   (*=================================================================================*)
   (* AM03_2   ---   Read Status + Send Control / Read Voltage + Current *)
   (*=================================================================================*)
   IF #Block2Size > 0 THEN
       // Read Total current and calculate it
       IF #C_Block2_TotalCurrent > 0 THEN
           (*Read Data*)
           #iError := DPRD_DAT(LADDR := #C_Block2_TotalCurrent, RECORD => #Current);
           (*Calculate Value*)
           #CalcValue := #Current[1];
           #CalcValue := SHL(IN := #CalcValue, N := 8);
           #O_Block2TotalCurrent := (#CalcValue + #Current[0]) / 100;
       END_IF;
       (*Status And Control*)
       IF #C_Block2_StatusControl > 0 THEN
           (*Read Inputs*)
           #iError := DPRD_DAT(LADDR := #C_Block2_StatusControl, RECORD => #Status);
           (*Take it over to the Datastructure*)
           FOR #iCount := 1 TO 32 DO
               IF #iCount <= #Block2Size * 2 THEN //WDL changed C_Block1Size by C_Block2Size
                   IF "SimulationActive" THEN
                       "NotUsedBool" := False;
                     ELSE
                       #IO_ETAFuseData.DataCPC20.Fuse[#iCount + 32].Status := #Status[#iCount]; (*Read Status*)
                   END_IF;
                   #Control[#iCount] := #IO_ETAFuseData.DataCPC20.Fuse[#iCount + 32].Control; (*Write control to the buffer*)
               ELSE
                   #IO_ETAFuseData.DataCPC20.Fuse[#iCount + 32].Status := 255; (*Read Status*)
                   #Control[#iCount] := 0; (*Write control to the buffer*)
               END_IF;
           END_FOR;
           (*Write outputs to the CPC*)
           #iError := DPWR_DAT(LADDR := #C_Block2_StatusControl, RECORD := #Control);
       END_IF;
       (*Measurement preperation*)
       IF #"C_Block2_MeasurementU/I" > 0 THEN
           (*Read measurenets values*)
           #iError := DPRD_DAT(LADDR := #"C_Block2_MeasurementU/I", RECORD => #UI);
           (*Create Measurements*)
           FOR #iCount := 1 TO 32 DO
               (*Calculate new Adress*)
               #iCalcAddress := ((#iCount - 1) * 4);
               IF #iCount <= #Block2Size * 2 THEN
                   (*Calculate current and take it over to the Datastructure*)
                   #CalcValue := #UI[#iCalcAddress + 1]; (*-2*)
                   #CalcValue := SHL(IN := #CalcValue, N := 8);
                   #IO_ETAFuseData.DataCPC20.Fuse[#iCount + 32].Current := INT_TO_REAL(#CalcValue + #UI[#iCalcAddress]) / 100; (*-3*)
                   (*Calculate voltage and take it over to the Datastructure*)
                   #CalcValue := #UI[#iCalcAddress + 3];
                   #CalcValue := SHL(IN := #CalcValue, N := 8); (*-0*)
                   #IO_ETAFuseData.DataCPC20.Fuse[#iCount + 32].Voltage := INT_TO_REAL(#CalcValue + #UI[#iCalcAddress + 2]) / 100; (*-1*)
               ELSE
                   #IO_ETAFuseData.DataCPC20.Fuse[#iCount + 32].Current := 0; (*-3*)
                   #IO_ETAFuseData.DataCPC20.Fuse[#iCount + 32].Voltage := 0; (*-1*)
               END_IF;
           END_FOR;
       END_IF;
   END_IF;

   (*=================================================================================*)
   (*AM03_1 & AM03_2   ---   Read Nominal Current *)    
   (*=================================================================================*)
   //HMI Command - Cancel Read nominal current
   IF #I_CancelReadNomCurr OR "SimulationActive" THEN
       #iCountGet := 1000;
   END_IF;

   CASE #iCountGet OF
       0: IF (#InitNominalCurrent OR #I_ReadNomCurr OR #I_NewShift) AND NOT #NonCyclicCommunication.ReadNomCurrActive AND NOT "SimulationActive" THEN
               IF (#C_Block1_TotalCurrent > 0) THEN
                   #iCountNominalCurrent := 1; // Init Value
                   #ChannelNumber := 1; // Init Value
                   #HardwareID := #C_Block1_TotalCurrent; // Init Value
                   #NonCyclicCommunication.ReadNomCurrActive := True;
                   #iCountGet := 10;
               END_IF;

               IF (#C_Block1_TotalCurrent = 0) AND (#C_Block2_TotalCurrent > 0) THEN
                   #iCountNominalCurrent := 33; // Init Value
                   #ChannelNumber := 1; // Init Value
                   #HardwareID := #C_Block2_TotalCurrent; // Init Value
                   #NonCyclicCommunication.ReadNomCurrActive := True;
                   #iCountGet := 10;
               END_IF;

               IF (#C_Block1_TotalCurrent = 0) AND (#C_Block2_TotalCurrent = 0) THEN
                   #Get.bGetData := False;
                   #iCountGet := 1000;
               END_IF;
           END_IF;
       10: // Set Parameter to read a channel and start it
           IF NOT #C_Config.Fuse[#iCountNominalCurrent].Used THEN
               #iCountNominalCurrent := #iCountNominalCurrent + 1;
               #ChannelNumber := #ChannelNumber + 1;
               #IO_ETAFuseData.DataCPC20.Fuse[#iCountNominalCurrent].NominalCurrent := 0;
               #iCountGet := 100;
           ELSE
               #Get.diIndex := (#ChannelNumber * 100) + 1; // Channel Number * Factor for Parameter + Index
               #Get.uiMlen := 8;
               #Get.bGetData := True; (*Read Data*)
               #iCountGet := 20;
           END_IF;

           IF (#iCountNominalCurrent >= 64) THEN
               #iCountGet := 1000;
           END_IF;
       20: (*reading is active*)
           IF #Get.bBusy OR #Get.bError THEN
               #Get.bGetData := false; (*Edge to read is enough*)
               #iCountGet := 30;
           END_IF;
       30: (*Evaluate data, stop reading, set message in case of error*)
           IF NOT #Get.bBusy THEN
               IF #Get.bValid THEN
                   #IO_ETAFuseData.DataCPC20.Fuse[#iCountNominalCurrent].NominalCurrent := #Get.DataByte[1] - 16#A0;
                   #iCountGet := 100;
               ELSE
                   #iCountGet := 10;
               END_IF;
           END_IF;
       100: // check for next channel
           IF (#iCountNominalCurrent >= 32) AND (#iCountNominalCurrent < 64) THEN
               #HardwareID := #C_Block2_TotalCurrent;
               #iCountNominalCurrent := #iCountNominalCurrent + 1;
               #ChannelNumber := #ChannelNumber + 1;
               #iCountGet := 10;
           END_IF;

           IF #iCountNominalCurrent < 32 THEN
               #HardwareID := #C_Block1_TotalCurrent;
               #iCountNominalCurrent := #iCountNominalCurrent + 1;
               #ChannelNumber := #ChannelNumber + 1;
               #iCountGet := 10;
           END_IF;

           IF (#iCountNominalCurrent = 33) THEN
               #ChannelNumber := 1;
           END_IF;

           IF (#iCountNominalCurrent >= 64) THEN
               #iCountGet := 1000;
           END_IF;
       1000: // End
           #InitNominalCurrent := False;
           #NonCyclicCommunication.ReadNomCurrActive := False;
           #iCountGet := 0;
   END_CASE;

   // Reading of nominal current is active
   #O_ReadNomCurrActive := #NonCyclicCommunication.ReadNomCurrActive;
   #O_ReadNomCurrFuseNr := #iCountNominalCurrent;

   // Overtime Reading of nominal current
   #T_ReadNomCurr(IN:= #O_ReadNomCurrActive,
                  PT:= T#60s);

   #O_AlarmReadNomCurr := #T_ReadNomCurr.Q;

   // Call noncyclic communication
   #RDREC_FB(REQ := #Get.bGetData,
             ID := #HardwareID,
             INDEX := #Get.diIndex,
             MLEN := #Get.uiMlen,
             VALID => #Get.bValid,
             BUSY => #Get.bBusy,
             ERROR => #Get.bError,
             STATUS => #Get.dwState,
             LEN => #Get.uilen,
             RECORD := #Get.DataByte);

   (*=================================================================================*)
   (* Fill-in/Clear Information *)    
   (*=================================================================================*)
   FOR #iCount := 1 TO 64 DO
       IF #C_Config.Fuse[#iCount].Used THEN
           #IO_ETAFuseData.ForHMICPC20.Fuse[#iCount].Used := True;
           #H_ETAFuseCPC20PN.H_ForHMI.ChannelInfo[#iCount].Name := #C_Config.Fuse[#iCount].Name;
           #H_ETAFuseCPC20PN.H_ForHMI.ChannelInfo[#iCount].Description := #C_Config.Fuse[#iCount].Description;
           #H_ETAFuseCPC20PN.H_ForHMI.ChannelInfo[#iCount].Current := #IO_ETAFuseData.DataCPC20.Fuse[#iCount].Current;
           #H_ETAFuseCPC20PN.H_ForHMI.ChannelInfo[#iCount].NominalCurrent := #IO_ETAFuseData.DataCPC20.Fuse[#iCount].NominalCurrent;
       ELSE
           #IO_ETAFuseData.DataCPC20.Fuse[#iCount] := #EmptyDataCPC20;
           #IO_ETAFuseData.DataCPC20.Fuse[#iCount].Status := 255;

           #IO_ETAFuseData.ForHMICPC20.Fuse[#iCount] := #EmptyForHMIFuse;

           #H_ETAFuseCPC20PN.H_ForHMI.Fuse[#iCount] := #EmptyForHMIFuse;
           #H_ETAFuseCPC20PN.H_ForHMI.ChannelInfo[#iCount] := #EmptyForHMIChannelInfo;
           #H_ETAFuseCPC20PN.H_ForHMI.ChannelInfo[#iCount].Name := 'Not exist';
       END_IF;
   END_FOR;

   #H_ETAFuseCPC20PN.H_ForHMI.Fuse := #IO_ETAFuseData.ForHMICPC20.Fuse;
END_FUNCTION_BLOCK

FUNCTION_BLOCK "L10Alarm"   // FB1410, FBD
TITLE = L10Alarm
{ S7_Optimized_Access := 'FALSE' }
AUTHOR : VCC
FAMILY : AlarmHnd
NAME : 10Alarm
VERSION : 1.0
// ================================================================================
// This module is used everywhere 10 alarms has to be generated when one 
// (security) corresponding input becomes True.
// All alarms can be True only when the corresponding input Enable Alarm is also 
// True.
// When the conditions to generate the alarm is disappear, a boolean (one per 
// alarm) available to inform the upper level that the corresponding alarm can be 
// reset. All alarms are reset by means of the AlarmResetPB signal.
// ================================================================================
// stored: AutoNumber false, IsIECCheckEnabled false, SetENOAutomatically False, UDAEnableTagReadback false
   VAR_INPUT
      I_Input1 { ExternalAccessible := 'False'; ExternalVisible := 'False'; ExternalWritable := 'False'} : Bool;   // Input alarm 1
      I_AlarmClass1 { ExternalAccessible := 'False'; ExternalVisible := 'False'; ExternalWritable := 'False'} : Char;   // Alarm class -> A - B - C - D or E
      I_EnableAlarm1 { ExternalAccessible := 'False'; ExternalVisible := 'False'; ExternalWritable := 'False'} : Bool := TRUE;   // Enable alarm 1 from upper level
      I_Invisible1 { ExternalAccessible := 'False'; ExternalVisible := 'False'; ExternalWritable := 'False'} : Bool;   // Invisible 1
      I_Input2 { ExternalAccessible := 'False'; ExternalVisible := 'False'; ExternalWritable := 'False'} : Bool;   // Input alarm 2
      I_AlarmClass2 { ExternalAccessible := 'False'; ExternalVisible := 'False'; ExternalWritable := 'False'} : Char;   // Alarm class -> A - B - C - D or E
      I_EnableAlarm2 { ExternalAccessible := 'False'; ExternalVisible := 'False'; ExternalWritable := 'False'} : Bool := TRUE;   // Enable alarm 2 from upper level
      I_Invisible2 { ExternalAccessible := 'False'; ExternalVisible := 'False'; ExternalWritable := 'False'} : Bool;   // Invisible 2
      I_Input3 { ExternalAccessible := 'False'; ExternalVisible := 'False'; ExternalWritable := 'False'} : Bool;   // Input alarm 3
      I_AlarmClass3 { ExternalAccessible := 'False'; ExternalVisible := 'False'; ExternalWritable := 'False'} : Char;   // Alarm class -> A - B - C - D or E
      I_EnableAlarm3 { ExternalAccessible := 'False'; ExternalVisible := 'False'; ExternalWritable := 'False'} : Bool := TRUE;   // Enable alarm 3 from upper level
      I_Invisible3 { ExternalAccessible := 'False'; ExternalVisible := 'False'; ExternalWritable := 'False'} : Bool;   // Invisible 3
      I_Input4 { ExternalAccessible := 'False'; ExternalVisible := 'False'; ExternalWritable := 'False'} : Bool;   // Input alarm 4
      I_AlarmClass4 { ExternalAccessible := 'False'; ExternalVisible := 'False'; ExternalWritable := 'False'} : Char;   // Alarm class -> A - B - C - D or E
      I_EnableAlarm4 { ExternalAccessible := 'False'; ExternalVisible := 'False'; ExternalWritable := 'False'} : Bool := TRUE;   // Enable alarm 4 from upper level
      I_Invisible4 { ExternalAccessible := 'False'; ExternalVisible := 'False'; ExternalWritable := 'False'} : Bool;   // Invisible 4
      I_Input5 { ExternalAccessible := 'False'; ExternalVisible := 'False'; ExternalWritable := 'False'} : Bool;   // Input alarm 5
      I_AlarmClass5 { ExternalAccessible := 'False'; ExternalVisible := 'False'; ExternalWritable := 'False'} : Char;   // Alarm class -> A - B - C - D or E
      I_EnableAlarm5 { ExternalAccessible := 'False'; ExternalVisible := 'False'; ExternalWritable := 'False'} : Bool := TRUE;   // Enable alarm 5 from upper level
      I_Invisible5 { ExternalAccessible := 'False'; ExternalVisible := 'False'; ExternalWritable := 'False'} : Bool;   // Invisible 5
      I_Input6 { ExternalAccessible := 'False'; ExternalVisible := 'False'; ExternalWritable := 'False'} : Bool;   // Input alarm 6
      I_AlarmClass6 { ExternalAccessible := 'False'; ExternalVisible := 'False'; ExternalWritable := 'False'} : Char;   // Alarm class -> A - B - C - D or E
      I_EnableAlarm6 { ExternalAccessible := 'False'; ExternalVisible := 'False'; ExternalWritable := 'False'} : Bool := TRUE;   // Enable alarm 6 from upper level
      I_Invisible6 { ExternalAccessible := 'False'; ExternalVisible := 'False'; ExternalWritable := 'False'} : Bool;   // Invisible 6
      I_Input7 { ExternalAccessible := 'False'; ExternalVisible := 'False'; ExternalWritable := 'False'} : Bool;   // Input alarm 7
      I_AlarmClass7 { ExternalAccessible := 'False'; ExternalVisible := 'False'; ExternalWritable := 'False'} : Char;   // Alarm class -> A - B - C - D or E
      I_EnableAlarm7 { ExternalAccessible := 'False'; ExternalVisible := 'False'; ExternalWritable := 'False'} : Bool := TRUE;   // Enable alarm 7 from upper level
      I_Invisible7 { ExternalAccessible := 'False'; ExternalVisible := 'False'; ExternalWritable := 'False'} : Bool;   // Invisible 7
      I_Input8 { ExternalAccessible := 'False'; ExternalVisible := 'False'; ExternalWritable := 'False'} : Bool;   // Input alarm 8
      I_AlarmClass8 { ExternalAccessible := 'False'; ExternalVisible := 'False'; ExternalWritable := 'False'} : Char;   // Alarm class -> A - B - C - D or E
      I_EnableAlarm8 { ExternalAccessible := 'False'; ExternalVisible := 'False'; ExternalWritable := 'False'} : Bool := TRUE;   // Enable alarm 8 from upper level
      I_Invisible8 { ExternalAccessible := 'False'; ExternalVisible := 'False'; ExternalWritable := 'False'} : Bool;   // Invisible 8
      I_Input9 { ExternalAccessible := 'False'; ExternalVisible := 'False'; ExternalWritable := 'False'} : Bool;   // Input alarm 9 (normally open)
      I_AlarmClass9 { ExternalAccessible := 'False'; ExternalVisible := 'False'; ExternalWritable := 'False'} : Char;   // Alarm class -> A - B - C - D or E
      I_EnableAlarm9 { ExternalAccessible := 'False'; ExternalVisible := 'False'; ExternalWritable := 'False'} : Bool := TRUE;   // Enable alarm 9 from upper level
      I_Invisible9 { ExternalAccessible := 'False'; ExternalVisible := 'False'; ExternalWritable := 'False'} : Bool;   // Invisible 9
      I_Input10 { ExternalAccessible := 'False'; ExternalVisible := 'False'; ExternalWritable := 'False'} : Bool;   // Input alarm 10
      I_AlarmClass10 { ExternalAccessible := 'False'; ExternalVisible := 'False'; ExternalWritable := 'False'} : Char;   // Alarm class -> A - B - C - D or E
      I_EnableAlarm10 { ExternalAccessible := 'False'; ExternalVisible := 'False'; ExternalWritable := 'False'} : Bool := TRUE;   // Enable alarm 10 from upper level
      I_Invisible10 { ExternalAccessible := 'False'; ExternalVisible := 'False'; ExternalWritable := 'False'} : Bool;   // Invisible 10
      I_AlarmResetPB { ExternalAccessible := 'False'; ExternalVisible := 'False'; ExternalWritable := 'False'} : Bool;   // Alarm reset pushbutton is activated
   END_VAR
   VAR_OUTPUT
      O_Alarm1 { ExternalAccessible := 'False'; ExternalVisible := 'False'; ExternalWritable := 'False'} : Bool;   // Alarm 1
      O_Alarm2 { ExternalAccessible := 'False'; ExternalVisible := 'False'; ExternalWritable := 'False'} : Bool;   // Alarm 2
      O_Alarm3 { ExternalAccessible := 'False'; ExternalVisible := 'False'; ExternalWritable := 'False'} : Bool;   // Alarm 3
      O_Alarm4 { ExternalAccessible := 'False'; ExternalVisible := 'False'; ExternalWritable := 'False'} : Bool;   // Alarm 4
      O_Alarm5 { ExternalAccessible := 'False'; ExternalVisible := 'False'; ExternalWritable := 'False'} : Bool;   // Alarm 5
      O_Alarm6 { ExternalAccessible := 'False'; ExternalVisible := 'False'; ExternalWritable := 'False'} : Bool;   // Alarm 6
      O_Alarm7 { ExternalAccessible := 'False'; ExternalVisible := 'False'; ExternalWritable := 'False'} : Bool;   // Alarm 7
      O_Alarm8 { ExternalAccessible := 'False'; ExternalVisible := 'False'; ExternalWritable := 'False'} : Bool;   // Alarm 8
      O_Alarm9 { ExternalAccessible := 'False'; ExternalVisible := 'False'; ExternalWritable := 'False'} : Bool;   // Alarm 9
      O_Alarm10 { ExternalAccessible := 'False'; ExternalVisible := 'False'; ExternalWritable := 'False'} : Bool;   // Alarm 10
      O_AlarmABCondition { ExternalAccessible := 'False'; ExternalVisible := 'False'; ExternalWritable := 'False'} : Bool;   // Alarm AB condition
      H_IAnim1 { ExternalAccessible := 'False'; ExternalVisible := 'False'; ExternalWritable := 'False'} : Word;   // Icon Animation 1
      H_IAnim2 { ExternalAccessible := 'False'; ExternalVisible := 'False'; ExternalWritable := 'False'} : Word;   // Icon Animation 2
      H_IAnim3 { ExternalAccessible := 'False'; ExternalVisible := 'False'; ExternalWritable := 'False'} : Word;   // Icon Animation 3
      H_IAnim4 { ExternalAccessible := 'False'; ExternalVisible := 'False'; ExternalWritable := 'False'} : Word;   // Icon Animation 4
      H_IAnim5 { ExternalAccessible := 'False'; ExternalVisible := 'False'; ExternalWritable := 'False'} : Word;   // Icon Animation 5
      H_IAnim6 { ExternalAccessible := 'False'; ExternalVisible := 'False'; ExternalWritable := 'False'} : Word;   // Icon Animation 6
      H_IAnim7 { ExternalAccessible := 'False'; ExternalVisible := 'False'; ExternalWritable := 'False'} : Word;   // Icon Animation 7
      H_IAnim8 { ExternalAccessible := 'False'; ExternalVisible := 'False'; ExternalWritable := 'False'} : Word;   // Icon Animation 8
      H_IAnim9 { ExternalAccessible := 'False'; ExternalVisible := 'False'; ExternalWritable := 'False'} : Word;   // Icon Animation 9
      H_IAnim10 { ExternalAccessible := 'False'; ExternalVisible := 'False'; ExternalWritable := 'False'} : Word;   // Icon Animation 10
   END_VAR
   VAR DB_SPECIFIC
      H_Out : Struct   // HMI
         Anim1 : Word;   // HMI Animation of the object
         Anim2 : Word;   // HMI Animation of the object
         Anim3 : Word;   // HMI Animation of the object
         Anim4 : Word;   // HMI Animation of the object
         Anim5 : Word;   // HMI Animation of the object
         Anim6 : Word;   // HMI Animation of the object
         Anim7 : Word;   // HMI Animation of the object
         Anim8 : Word;   // HMI Animation of the object
         Anim9 : Word;   // HMI Animation of the object
         Anim10 : Word;   // HMI Animation of the object
         DBnr : Int;   // HMI Animation DB number
      END_STRUCT;
      Alarm1 { ExternalAccessible := 'False'; ExternalVisible := 'False'; ExternalWritable := 'False'} : Bool;   // Alarm 1
      AlarmClass1_A { ExternalAccessible := 'False'; ExternalVisible := 'False'; ExternalWritable := 'False'} : Bool;   // The alarm is from alarm class A
      AlarmClass1_B { ExternalAccessible := 'False'; ExternalVisible := 'False'; ExternalWritable := 'False'} : Bool;   // The alarm is from alarm class B
      AlarmClass1_C { ExternalAccessible := 'False'; ExternalVisible := 'False'; ExternalWritable := 'False'} : Bool;   // The alarm is from alarm class C
      AlarmClass1_D { ExternalAccessible := 'False'; ExternalVisible := 'False'; ExternalWritable := 'False'} : Bool;   // The alarm is from alarm class D
      AlarmClass1_E { ExternalAccessible := 'False'; ExternalVisible := 'False'; ExternalWritable := 'False'} : Bool;   // The alarm is from alarm class E
      Alarm1Cond { ExternalAccessible := 'False'; ExternalVisible := 'False'; ExternalWritable := 'False'} : Bool;   // Alarm 1 condition
      Alarm2 { ExternalAccessible := 'False'; ExternalVisible := 'False'; ExternalWritable := 'False'} : Bool;   // Alarm 2
      AlarmClass2_A { ExternalAccessible := 'False'; ExternalVisible := 'False'; ExternalWritable := 'False'} : Bool;   // The alarm is from alarm class A
      AlarmClass2_B { ExternalAccessible := 'False'; ExternalVisible := 'False'; ExternalWritable := 'False'} : Bool;   // The alarm is from alarm class B
      AlarmClass2_C { ExternalAccessible := 'False'; ExternalVisible := 'False'; ExternalWritable := 'False'} : Bool;   // The alarm is from alarm class C
      AlarmClass2_D { ExternalAccessible := 'False'; ExternalVisible := 'False'; ExternalWritable := 'False'} : Bool;   // The alarm is from alarm class D
      AlarmClass2_E { ExternalAccessible := 'False'; ExternalVisible := 'False'; ExternalWritable := 'False'} : Bool;   // The alarm is from alarm class E
      Alarm2Cond { ExternalAccessible := 'False'; ExternalVisible := 'False'; ExternalWritable := 'False'} : Bool;   // Alarm 2 condition
      Alarm3 { ExternalAccessible := 'False'; ExternalVisible := 'False'; ExternalWritable := 'False'} : Bool;   // Alarm 3
      AlarmClass3_A { ExternalAccessible := 'False'; ExternalVisible := 'False'; ExternalWritable := 'False'} : Bool;   // The alarm is from alarm class A
      AlarmClass3_B { ExternalAccessible := 'False'; ExternalVisible := 'False'; ExternalWritable := 'False'} : Bool;   // The alarm is from alarm class B
      AlarmClass3_C { ExternalAccessible := 'False'; ExternalVisible := 'False'; ExternalWritable := 'False'} : Bool;   // The alarm is from alarm class C
      AlarmClass3_D { ExternalAccessible := 'False'; ExternalVisible := 'False'; ExternalWritable := 'False'} : Bool;   // The alarm is from alarm class D
      AlarmClass3_E { ExternalAccessible := 'False'; ExternalVisible := 'False'; ExternalWritable := 'False'} : Bool;   // The alarm is from alarm class E
      Alarm3Cond { ExternalAccessible := 'False'; ExternalVisible := 'False'; ExternalWritable := 'False'} : Bool;   // Alarm 3 condition
      Alarm4 { ExternalAccessible := 'False'; ExternalVisible := 'False'; ExternalWritable := 'False'} : Bool;   // Alarm 4
      AlarmClass4_A { ExternalAccessible := 'False'; ExternalVisible := 'False'; ExternalWritable := 'False'} : Bool;   // The alarm is from alarm class A
      AlarmClass4_B { ExternalAccessible := 'False'; ExternalVisible := 'False'; ExternalWritable := 'False'} : Bool;   // The alarm is from alarm class B
      AlarmClass4_C { ExternalAccessible := 'False'; ExternalVisible := 'False'; ExternalWritable := 'False'} : Bool;   // The alarm is from alarm class C
      AlarmClass4_D { ExternalAccessible := 'False'; ExternalVisible := 'False'; ExternalWritable := 'False'} : Bool;   // The alarm is from alarm class D
      AlarmClass4_E { ExternalAccessible := 'False'; ExternalVisible := 'False'; ExternalWritable := 'False'} : Bool;   // The alarm is from alarm class E
      Alarm4Cond { ExternalAccessible := 'False'; ExternalVisible := 'False'; ExternalWritable := 'False'} : Bool;   // Alarm 4 condition
      Alarm5 { ExternalAccessible := 'False'; ExternalVisible := 'False'; ExternalWritable := 'False'} : Bool;   // Alarm 5
      AlarmClass5_A { ExternalAccessible := 'False'; ExternalVisible := 'False'; ExternalWritable := 'False'} : Bool;   // The alarm is from alarm class A
      AlarmClass5_B { ExternalAccessible := 'False'; ExternalVisible := 'False'; ExternalWritable := 'False'} : Bool;   // The alarm is from alarm class B
      AlarmClass5_C { ExternalAccessible := 'False'; ExternalVisible := 'False'; ExternalWritable := 'False'} : Bool;   // The alarm is from alarm class C
      AlarmClass5_D { ExternalAccessible := 'False'; ExternalVisible := 'False'; ExternalWritable := 'False'} : Bool;   // The alarm is from alarm class D
      AlarmClass5_E { ExternalAccessible := 'False'; ExternalVisible := 'False'; ExternalWritable := 'False'} : Bool;   // The alarm is from alarm class E
      Alarm5Cond { ExternalAccessible := 'False'; ExternalVisible := 'False'; ExternalWritable := 'False'} : Bool;   // Alarm 5 condition
      Alarm6 { ExternalAccessible := 'False'; ExternalVisible := 'False'; ExternalWritable := 'False'} : Bool;   // Alarm 6
      AlarmClass6_A { ExternalAccessible := 'False'; ExternalVisible := 'False'; ExternalWritable := 'False'} : Bool;   // The alarm is from alarm class A
      AlarmClass6_B { ExternalAccessible := 'False'; ExternalVisible := 'False'; ExternalWritable := 'False'} : Bool;   // The alarm is from alarm class B
      AlarmClass6_C { ExternalAccessible := 'False'; ExternalVisible := 'False'; ExternalWritable := 'False'} : Bool;   // The alarm is from alarm class C
      AlarmClass6_D { ExternalAccessible := 'False'; ExternalVisible := 'False'; ExternalWritable := 'False'} : Bool;   // The alarm is from alarm class D
      AlarmClass6_E { ExternalAccessible := 'False'; ExternalVisible := 'False'; ExternalWritable := 'False'} : Bool;   // The alarm is from alarm class E
      Alarm6Cond { ExternalAccessible := 'False'; ExternalVisible := 'False'; ExternalWritable := 'False'} : Bool;   // Alarm 6 condition
      Alarm7 { ExternalAccessible := 'False'; ExternalVisible := 'False'; ExternalWritable := 'False'} : Bool;   // Alarm 7
      AlarmClass7_A { ExternalAccessible := 'False'; ExternalVisible := 'False'; ExternalWritable := 'False'} : Bool;   // The alarm is from alarm class A
      AlarmClass7_B { ExternalAccessible := 'False'; ExternalVisible := 'False'; ExternalWritable := 'False'} : Bool;   // The alarm is from alarm class B
      AlarmClass7_C { ExternalAccessible := 'False'; ExternalVisible := 'False'; ExternalWritable := 'False'} : Bool;   // The alarm is from alarm class C
      AlarmClass7_D { ExternalAccessible := 'False'; ExternalVisible := 'False'; ExternalWritable := 'False'} : Bool;   // The alarm is from alarm class D
      AlarmClass7_E { ExternalAccessible := 'False'; ExternalVisible := 'False'; ExternalWritable := 'False'} : Bool;   // The alarm is from alarm class E
      Alarm7Cond { ExternalAccessible := 'False'; ExternalVisible := 'False'; ExternalWritable := 'False'} : Bool;   // Alarm 7 condition
      Alarm8 { ExternalAccessible := 'False'; ExternalVisible := 'False'; ExternalWritable := 'False'} : Bool;   // Alarm 8
      AlarmClass8_A { ExternalAccessible := 'False'; ExternalVisible := 'False'; ExternalWritable := 'False'} : Bool;   // The alarm is from alarm class A
      AlarmClass8_B { ExternalAccessible := 'False'; ExternalVisible := 'False'; ExternalWritable := 'False'} : Bool;   // The alarm is from alarm class B
      AlarmClass8_C { ExternalAccessible := 'False'; ExternalVisible := 'False'; ExternalWritable := 'False'} : Bool;   // The alarm is from alarm class C
      AlarmClass8_D { ExternalAccessible := 'False'; ExternalVisible := 'False'; ExternalWritable := 'False'} : Bool;   // The alarm is from alarm class D
      AlarmClass8_E { ExternalAccessible := 'False'; ExternalVisible := 'False'; ExternalWritable := 'False'} : Bool;   // The alarm is from alarm class E
      Alarm8Cond { ExternalAccessible := 'False'; ExternalVisible := 'False'; ExternalWritable := 'False'} : Bool;   // Alarm 8 condition
      Alarm9 { ExternalAccessible := 'False'; ExternalVisible := 'False'; ExternalWritable := 'False'} : Bool;   // Alarm 9
      AlarmClass9_A { ExternalAccessible := 'False'; ExternalVisible := 'False'; ExternalWritable := 'False'} : Bool;   // The alarm is from alarm class A
      AlarmClass9_B { ExternalAccessible := 'False'; ExternalVisible := 'False'; ExternalWritable := 'False'} : Bool;   // The alarm is from alarm class B
      AlarmClass9_C { ExternalAccessible := 'False'; ExternalVisible := 'False'; ExternalWritable := 'False'} : Bool;   // The alarm is from alarm class C
      AlarmClass9_D { ExternalAccessible := 'False'; ExternalVisible := 'False'; ExternalWritable := 'False'} : Bool;   // The alarm is from alarm class D
      AlarmClass9_E { ExternalAccessible := 'False'; ExternalVisible := 'False'; ExternalWritable := 'False'} : Bool;   // The alarm is from alarm class E
      Alarm9Cond { ExternalAccessible := 'False'; ExternalVisible := 'False'; ExternalWritable := 'False'} : Bool;   // Alarm 9 condition
      Alarm10 { ExternalAccessible := 'False'; ExternalVisible := 'False'; ExternalWritable := 'False'} : Bool;   // Alarm 10
      AlarmClass10_A { ExternalAccessible := 'False'; ExternalVisible := 'False'; ExternalWritable := 'False'} : Bool;   // The alarm is from alarm class A
      AlarmClass10_B { ExternalAccessible := 'False'; ExternalVisible := 'False'; ExternalWritable := 'False'} : Bool;   // The alarm is from alarm class B
      AlarmClass10_C { ExternalAccessible := 'False'; ExternalVisible := 'False'; ExternalWritable := 'False'} : Bool;   // The alarm is from alarm class C
      AlarmClass10_D { ExternalAccessible := 'False'; ExternalVisible := 'False'; ExternalWritable := 'False'} : Bool;   // The alarm is from alarm class D
      AlarmClass10_E { ExternalAccessible := 'False'; ExternalVisible := 'False'; ExternalWritable := 'False'} : Bool;   // The alarm is from alarm class E
      Alarm10Cond { ExternalAccessible := 'False'; ExternalVisible := 'False'; ExternalWritable := 'False'} : Bool;   // Alarm 10 condition
      DBnr { ExternalAccessible := 'False'; ExternalVisible := 'False'; ExternalWritable := 'False'} : Int;   // HMI DB number
   END_VAR
BEGIN

NETWORK
TITLE = **** 1 - Inputs **** DB number
// DB number
      L     DINO;
      T     #DBnr;

NETWORK
TITLE = **** 1 - Inputs **** Alarm class 1
// Alarm class
// Alarm class = E
      L     #I_AlarmClass1;
      L     'E';
      ==I;
      =     #AlarmClass1_E;

// Alarm class = D
      L     #I_AlarmClass1;
      L     'D';
      ==I;
      =     #AlarmClass1_D;

// Alarm class = C
      L     #I_AlarmClass1;
      L     'C';
      ==I;
      =     #AlarmClass1_C;

// Alarm class = B
      L     #I_AlarmClass1;
      L     'B';
      ==I;
      =     #AlarmClass1_B;

// Alarm class = A
      AN    #AlarmClass1_B;
      AN    #AlarmClass1_C;
      AN    #AlarmClass1_D;
      AN    #AlarmClass1_E;
      =     #AlarmClass1_A;


NETWORK
TITLE = **** 1 - Inputs **** Alarm class 2
// Alarm class
// Alarm class = E
      L     #I_AlarmClass2;
      L     'E';
      ==I;
      =     #AlarmClass2_E;

// Alarm class = D
      L     #I_AlarmClass2;
      L     'D';
      ==I;
      =     #AlarmClass2_D;

// Alarm class = C
      L     #I_AlarmClass2;
      L     'C';
      ==I;
      =     #AlarmClass2_C;

// Alarm class = B
      L     #I_AlarmClass2;
      L     'B';
      ==I;
      =     #AlarmClass2_B;

// Alarm class = A
      AN    #AlarmClass2_B;
      AN    #AlarmClass2_C;
      AN    #AlarmClass2_D;
      AN    #AlarmClass2_E;
      =     #AlarmClass2_A;


NETWORK
TITLE = **** 1 - Inputs **** Alarm class 3
// Alarm class
// Alarm class = E
      L     #I_AlarmClass3;
      L     'E';
      ==I;
      =     #AlarmClass3_E;

// Alarm class = D
      L     #I_AlarmClass3;
      L     'D';
      ==I;
      =     #AlarmClass3_D;

// Alarm class = C
      L     #I_AlarmClass3;
      L     'C';
      ==I;
      =     #AlarmClass3_C;

// Alarm class = B
      L     #I_AlarmClass3;
      L     'B';
      ==I;
      =     #AlarmClass3_B;

// Alarm class = A
      AN    #AlarmClass3_B;
      AN    #AlarmClass3_C;
      AN    #AlarmClass3_D;
      AN    #AlarmClass3_E;
      =     #AlarmClass3_A;


NETWORK
TITLE = **** 1 - Inputs **** Alarm class 4
// Alarm class
// Alarm class = E
      L     #I_AlarmClass4;
      L     'E';
      ==I;
      =     #AlarmClass4_E;

// Alarm class = D
      L     #I_AlarmClass4;
      L     'D';
      ==I;
      =     #AlarmClass4_D;

// Alarm class = C
      L     #I_AlarmClass4;
      L     'C';
      ==I;
      =     #AlarmClass4_C;

// Alarm class = B
      L     #I_AlarmClass4;
      L     'B';
      ==I;
      =     #AlarmClass4_B;

// Alarm class = A
      AN    #AlarmClass4_B;
      AN    #AlarmClass4_C;
      AN    #AlarmClass4_D;
      AN    #AlarmClass4_E;
      =     #AlarmClass4_A;


NETWORK
TITLE = **** 1 - Inputs **** Alarm class 5
// Alarm class
// Alarm class = E
      L     #I_AlarmClass5;
      L     'E';
      ==I;
      =     #AlarmClass5_E;

// Alarm class = D
      L     #I_AlarmClass5;
      L     'D';
      ==I;
      =     #AlarmClass5_D;

// Alarm class = C
      L     #I_AlarmClass5;
      L     'C';
      ==I;
      =     #AlarmClass5_C;

// Alarm class = B
      L     #I_AlarmClass5;
      L     'B';
      ==I;
      =     #AlarmClass5_B;

// Alarm class = A
      AN    #AlarmClass5_B;
      AN    #AlarmClass5_C;
      AN    #AlarmClass5_D;
      AN    #AlarmClass5_E;
      =     #AlarmClass5_A;


NETWORK
TITLE = **** 1 - Inputs **** Alarm class 6
// Alarm class
// Alarm class = E
      L     #I_AlarmClass6;
      L     'E';
      ==I;
      =     #AlarmClass6_E;

// Alarm class = D
      L     #I_AlarmClass6;
      L     'D';
      ==I;
      =     #AlarmClass6_D;

// Alarm class = C
      L     #I_AlarmClass6;
      L     'C';
      ==I;
      =     #AlarmClass6_C;

// Alarm class = B
      L     #I_AlarmClass6;
      L     'B';
      ==I;
      =     #AlarmClass6_B;

// Alarm class = A
      AN    #AlarmClass6_B;
      AN    #AlarmClass6_C;
      AN    #AlarmClass6_D;
      AN    #AlarmClass6_E;
      =     #AlarmClass6_A;


NETWORK
TITLE = **** 1 - Inputs **** Alarm class 7
// Alarm class
// Alarm class = E
      L     #I_AlarmClass7;
      L     'E';
      ==I;
      =     #AlarmClass7_E;

// Alarm class = D
      L     #I_AlarmClass7;
      L     'D';
      ==I;
      =     #AlarmClass7_D;

// Alarm class = C
      L     #I_AlarmClass7;
      L     'C';
      ==I;
      =     #AlarmClass7_C;

// Alarm class = B
      L     #I_AlarmClass7;
      L     'B';
      ==I;
      =     #AlarmClass7_B;

// Alarm class = A
      AN    #AlarmClass7_B;
      AN    #AlarmClass7_C;
      AN    #AlarmClass7_D;
      AN    #AlarmClass7_E;
      =     #AlarmClass7_A;


NETWORK
TITLE = **** 1 - Inputs **** Alarm class 8
// Alarm class
// Alarm class = E
      L     #I_AlarmClass8;
      L     'E';
      ==I;
      =     #AlarmClass8_E;

// Alarm class = D
      L     #I_AlarmClass8;
      L     'D';
      ==I;
      =     #AlarmClass8_D;

// Alarm class = C
      L     #I_AlarmClass8;
      L     'C';
      ==I;
      =     #AlarmClass8_C;

// Alarm class = B
      L     #I_AlarmClass8;
      L     'B';
      ==I;
      =     #AlarmClass8_B;

// Alarm class = A
      AN    #AlarmClass8_B;
      AN    #AlarmClass8_C;
      AN    #AlarmClass8_D;
      AN    #AlarmClass8_E;
      =     #AlarmClass8_A;


NETWORK
TITLE = **** 1 - Inputs **** Alarm class 9
// Alarm class
// Alarm class = E
      L     #I_AlarmClass9;
      L     'E';
      ==I;
      =     #AlarmClass9_E;

// Alarm class = D
      L     #I_AlarmClass9;
      L     'D';
      ==I;
      =     #AlarmClass9_D;

// Alarm class = C
      L     #I_AlarmClass9;
      L     'C';
      ==I;
      =     #AlarmClass9_C;

// Alarm class = B
      L     #I_AlarmClass9;
      L     'B';
      ==I;
      =     #AlarmClass9_B;

// Alarm class = A
      AN    #AlarmClass9_B;
      AN    #AlarmClass9_C;
      AN    #AlarmClass9_D;
      AN    #AlarmClass9_E;
      =     #AlarmClass9_A;


NETWORK
TITLE = **** 1 - Inputs **** Alarm class 10
// Alarm class
// Alarm class = E
      L     #I_AlarmClass10;
      L     'E';
      ==I;
      =     #AlarmClass10_E;

// Alarm class = D
      L     #I_AlarmClass10;
      L     'D';
      ==I;
      =     #AlarmClass10_D;

// Alarm class = C
      L     #I_AlarmClass10;
      L     'C';
      ==I;
      =     #AlarmClass10_C;

// Alarm class = B
      L     #I_AlarmClass10;
      L     'B';
      ==I;
      =     #AlarmClass10_B;

// Alarm class = A
      AN    #AlarmClass10_B;
      AN    #AlarmClass10_C;
      AN    #AlarmClass10_D;
      AN    #AlarmClass10_E;
      =     #AlarmClass10_A;


REGION Network 12: **** 2.2 - Alarms - Alarms Generation **** Alarm Condition 1
   // Condition for Alarm 1
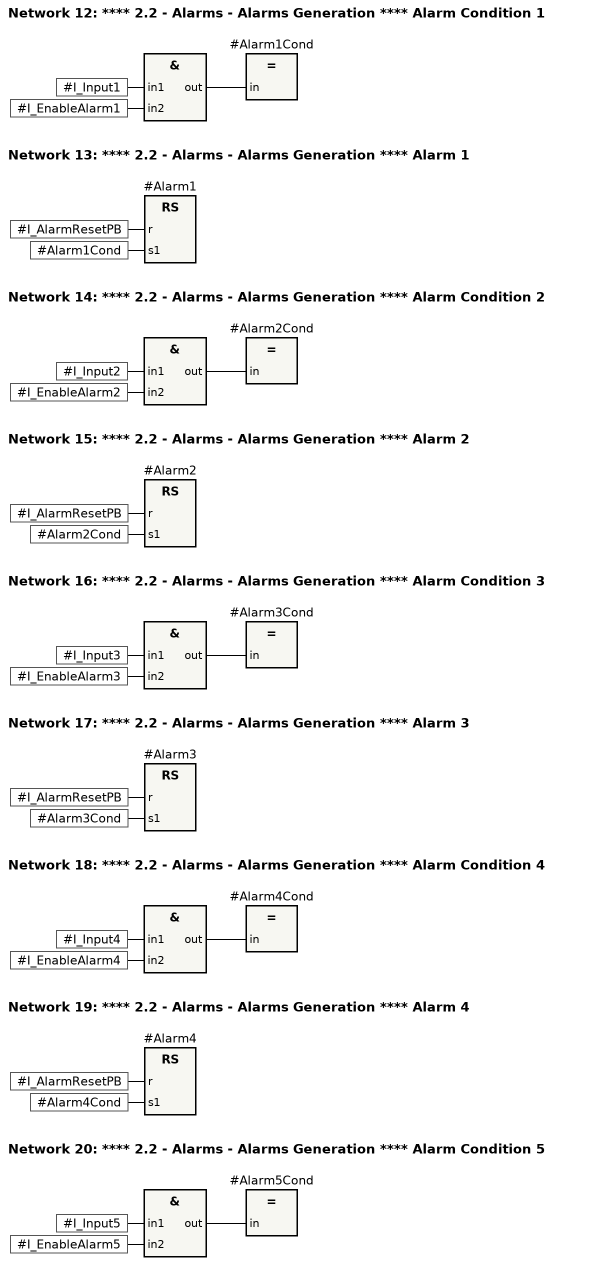
   #Alarm1Cond := #I_Input1 AND #I_EnableAlarm1;
END_REGION

REGION Network 13: **** 2.2 - Alarms - Alarms Generation **** Alarm 1
   // Creation of the Alarm 1
   IF #I_AlarmResetPB THEN
       #Alarm1 := FALSE;   // RS flip-flop
   END_IF;
   IF #Alarm1Cond THEN #Alarm1 := TRUE; END_IF;
END_REGION

REGION Network 14: **** 2.2 - Alarms - Alarms Generation **** Alarm Condition 2
   // Condition for Alarm 2
   #Alarm2Cond := #I_Input2 AND #I_EnableAlarm2;
END_REGION

REGION Network 15: **** 2.2 - Alarms - Alarms Generation **** Alarm 2
   // Creation of the Alarm 2
   IF #I_AlarmResetPB THEN
       #Alarm2 := FALSE;   // RS flip-flop
   END_IF;
   IF #Alarm2Cond THEN #Alarm2 := TRUE; END_IF;
END_REGION

REGION Network 16: **** 2.2 - Alarms - Alarms Generation **** Alarm Condition 3
   // Condition for Alarm 3
   #Alarm3Cond := #I_Input3 AND #I_EnableAlarm3;
END_REGION

REGION Network 17: **** 2.2 - Alarms - Alarms Generation **** Alarm 3
   // Creation of the Alarm 3
   IF #I_AlarmResetPB THEN
       #Alarm3 := FALSE;   // RS flip-flop
   END_IF;
   IF #Alarm3Cond THEN #Alarm3 := TRUE; END_IF;
END_REGION

REGION Network 18: **** 2.2 - Alarms - Alarms Generation **** Alarm Condition 4
   // Condition for Alarm 4
   #Alarm4Cond := #I_Input4 AND #I_EnableAlarm4;
END_REGION

REGION Network 19: **** 2.2 - Alarms - Alarms Generation **** Alarm 4
   // Creation of the Alarm 4
   IF #I_AlarmResetPB THEN
       #Alarm4 := FALSE;   // RS flip-flop
   END_IF;
   IF #Alarm4Cond THEN #Alarm4 := TRUE; END_IF;
END_REGION

REGION Network 20: **** 2.2 - Alarms - Alarms Generation **** Alarm Condition 5
   // Condition for Alarm 5
   #Alarm5Cond := #I_Input5 AND #I_EnableAlarm5;
END_REGION

REGION Network 21: **** 2.2 - Alarms - Alarms Generation **** Alarm 5
   // Creation of the Alarm 5
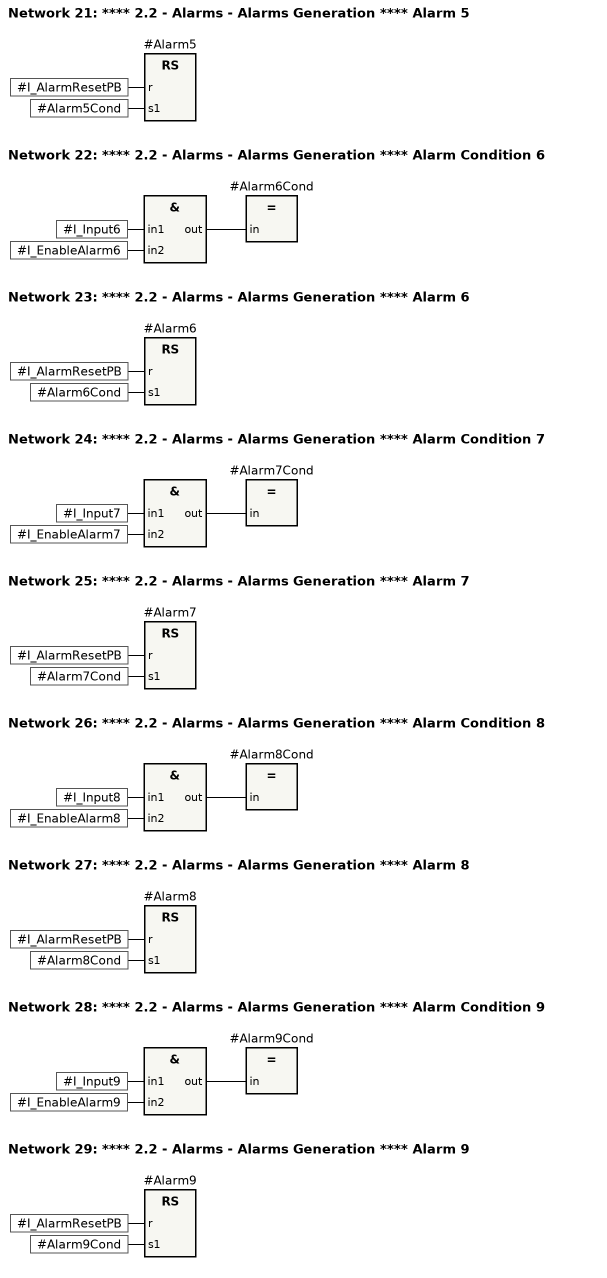
   IF #I_AlarmResetPB THEN
       #Alarm5 := FALSE;   // RS flip-flop
   END_IF;
   IF #Alarm5Cond THEN #Alarm5 := TRUE; END_IF;
END_REGION

REGION Network 22: **** 2.2 - Alarms - Alarms Generation **** Alarm Condition 6
   // Condition for Alarm 6
   #Alarm6Cond := #I_Input6 AND #I_EnableAlarm6;
END_REGION

REGION Network 23: **** 2.2 - Alarms - Alarms Generation **** Alarm 6
   // Creation of the Alarm 6
   IF #I_AlarmResetPB THEN
       #Alarm6 := FALSE;   // RS flip-flop
   END_IF;
   IF #Alarm6Cond THEN #Alarm6 := TRUE; END_IF;
END_REGION

REGION Network 24: **** 2.2 - Alarms - Alarms Generation **** Alarm Condition 7
   // Condition for Alarm 7
   #Alarm7Cond := #I_Input7 AND #I_EnableAlarm7;
END_REGION

REGION Network 25: **** 2.2 - Alarms - Alarms Generation **** Alarm 7
   // Creation of the Alarm 7
   IF #I_AlarmResetPB THEN
       #Alarm7 := FALSE;   // RS flip-flop
   END_IF;
   IF #Alarm7Cond THEN #Alarm7 := TRUE; END_IF;
END_REGION

REGION Network 26: **** 2.2 - Alarms - Alarms Generation **** Alarm Condition 8
   // Condition for Alarm 8
   #Alarm8Cond := #I_Input8 AND #I_EnableAlarm8;
END_REGION

REGION Network 27: **** 2.2 - Alarms - Alarms Generation **** Alarm 8
   // Creation of the Alarm 8
   IF #I_AlarmResetPB THEN
       #Alarm8 := FALSE;   // RS flip-flop
   END_IF;
   IF #Alarm8Cond THEN #Alarm8 := TRUE; END_IF;
END_REGION

REGION Network 28: **** 2.2 - Alarms - Alarms Generation **** Alarm Condition 9
   // Condition for Alarm 9
   #Alarm9Cond := #I_Input9 AND #I_EnableAlarm9;
END_REGION

REGION Network 29: **** 2.2 - Alarms - Alarms Generation **** Alarm 9
   // Creation of the Alarm 9
   IF #I_AlarmResetPB THEN
       #Alarm9 := FALSE;   // RS flip-flop
   END_IF;
   IF #Alarm9Cond THEN #Alarm9 := TRUE; END_IF;
END_REGION

REGION Network 30: **** 2.2 - Alarms - Alarms Generation **** Alarm Condition 10
   // Condition for Alarm 10
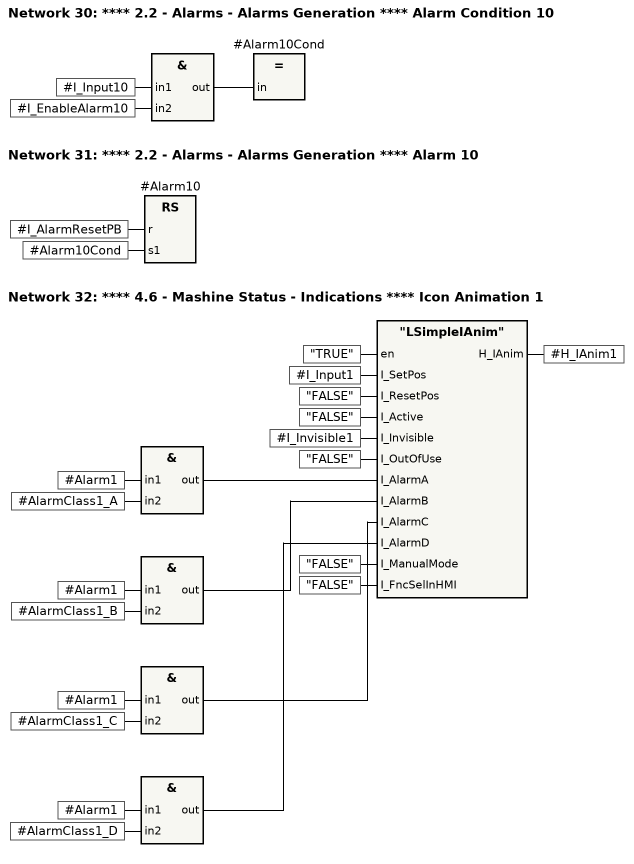
   #Alarm10Cond := #I_Input10 AND #I_EnableAlarm10;
END_REGION

REGION Network 31: **** 2.2 - Alarms - Alarms Generation **** Alarm 10
   // Creation of the Alarm 10
   IF #I_AlarmResetPB THEN
       #Alarm10 := FALSE;   // RS flip-flop
   END_IF;
   IF #Alarm10Cond THEN #Alarm10 := TRUE; END_IF;
END_REGION

REGION Network 32: **** 4.6 - Mashine Status - Indications **** Icon Animation 1
   // Icon Animation 1
   IF "TRUE" THEN
       "LSimpleIAnim"(I_SetPos := #I_Input1,
                      I_ResetPos := "FALSE",
                      I_Active := "FALSE",
                      I_Invisible := #I_Invisible1,
                      I_OutOfUse := "FALSE",
                      I_AlarmA := #Alarm1 AND #AlarmClass1_A,
                      I_AlarmB := #Alarm1 AND #AlarmClass1_B,
                      I_AlarmC := #Alarm1 AND #AlarmClass1_C,
                      I_AlarmD := #Alarm1 AND #AlarmClass1_D,
                      I_ManualMode := "FALSE",
                      I_FncSelInHMI := "FALSE",
                      H_IAnim => #H_IAnim1);
   END_IF;
END_REGION

REGION Network 33: **** 4.6 - Mashine Status - Indications **** Icon Animation 2
   // Icon Animation 2
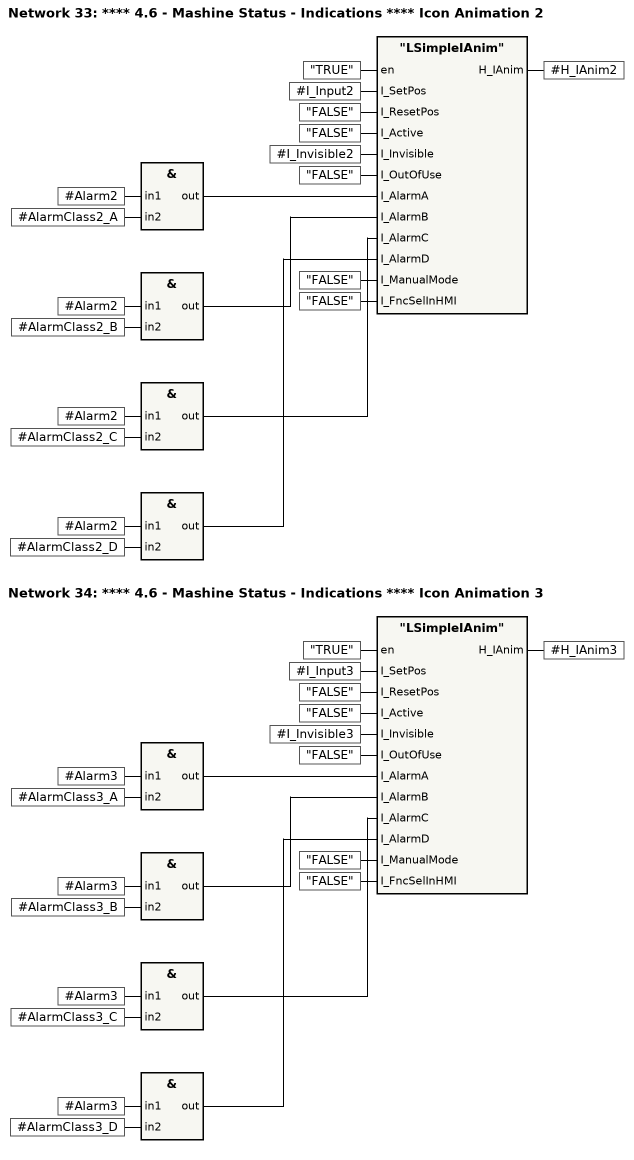
   IF "TRUE" THEN
       "LSimpleIAnim"(I_SetPos := #I_Input2,
                      I_ResetPos := "FALSE",
                      I_Active := "FALSE",
                      I_Invisible := #I_Invisible2,
                      I_OutOfUse := "FALSE",
                      I_AlarmA := #Alarm2 AND #AlarmClass2_A,
                      I_AlarmB := #Alarm2 AND #AlarmClass2_B,
                      I_AlarmC := #Alarm2 AND #AlarmClass2_C,
                      I_AlarmD := #Alarm2 AND #AlarmClass2_D,
                      I_ManualMode := "FALSE",
                      I_FncSelInHMI := "FALSE",
                      H_IAnim => #H_IAnim2);
   END_IF;
END_REGION

REGION Network 34: **** 4.6 - Mashine Status - Indications **** Icon Animation 3
   // Icon Animation 3
   IF "TRUE" THEN
       "LSimpleIAnim"(I_SetPos := #I_Input3,
                      I_ResetPos := "FALSE",
                      I_Active := "FALSE",
                      I_Invisible := #I_Invisible3,
                      I_OutOfUse := "FALSE",
                      I_AlarmA := #Alarm3 AND #AlarmClass3_A,
                      I_AlarmB := #Alarm3 AND #AlarmClass3_B,
                      I_AlarmC := #Alarm3 AND #AlarmClass3_C,
                      I_AlarmD := #Alarm3 AND #AlarmClass3_D,
                      I_ManualMode := "FALSE",
                      I_FncSelInHMI := "FALSE",
                      H_IAnim => #H_IAnim3);
   END_IF;
END_REGION

REGION Network 35: **** 4.6 - Mashine Status - Indications **** Icon Animation 4
   // Icon Animation 4
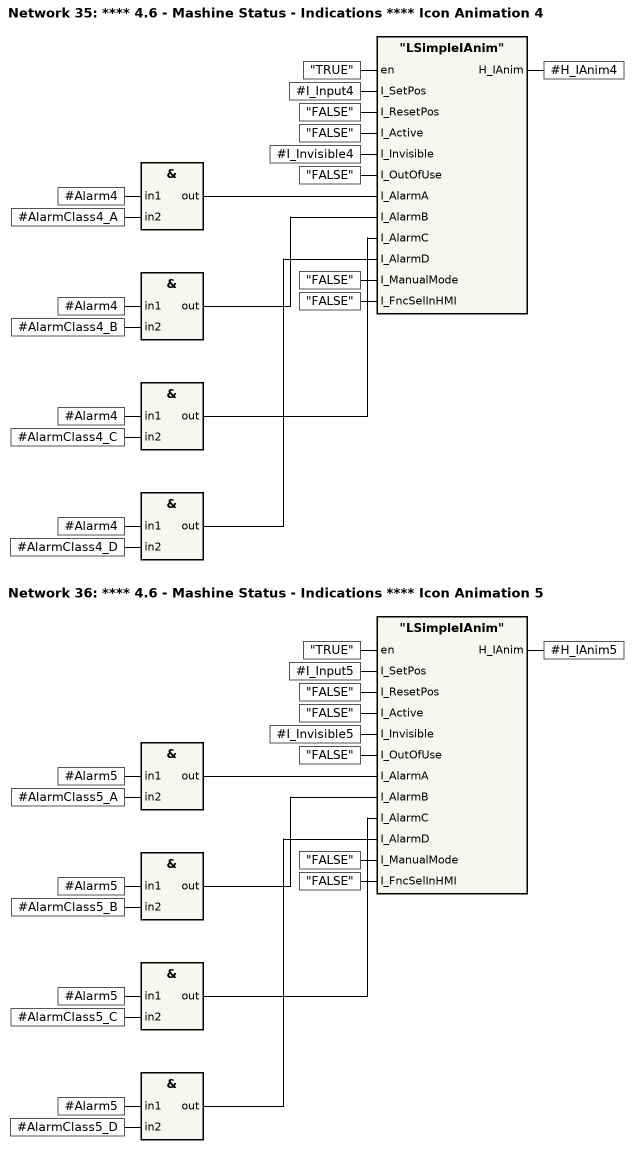
   IF "TRUE" THEN
       "LSimpleIAnim"(I_SetPos := #I_Input4,
                      I_ResetPos := "FALSE",
                      I_Active := "FALSE",
                      I_Invisible := #I_Invisible4,
                      I_OutOfUse := "FALSE",
                      I_AlarmA := #Alarm4 AND #AlarmClass4_A,
                      I_AlarmB := #Alarm4 AND #AlarmClass4_B,
                      I_AlarmC := #Alarm4 AND #AlarmClass4_C,
                      I_AlarmD := #Alarm4 AND #AlarmClass4_D,
                      I_ManualMode := "FALSE",
                      I_FncSelInHMI := "FALSE",
                      H_IAnim => #H_IAnim4);
   END_IF;
END_REGION

REGION Network 36: **** 4.6 - Mashine Status - Indications **** Icon Animation 5
   // Icon Animation 5
   IF "TRUE" THEN
       "LSimpleIAnim"(I_SetPos := #I_Input5,
                      I_ResetPos := "FALSE",
                      I_Active := "FALSE",
                      I_Invisible := #I_Invisible5,
                      I_OutOfUse := "FALSE",
                      I_AlarmA := #Alarm5 AND #AlarmClass5_A,
                      I_AlarmB := #Alarm5 AND #AlarmClass5_B,
                      I_AlarmC := #Alarm5 AND #AlarmClass5_C,
                      I_AlarmD := #Alarm5 AND #AlarmClass5_D,
                      I_ManualMode := "FALSE",
                      I_FncSelInHMI := "FALSE",
                      H_IAnim => #H_IAnim5);
   END_IF;
END_REGION

REGION Network 37: **** 4.6 - Mashine Status - Indications **** Icon Animation 6
   // Icon Animation 6
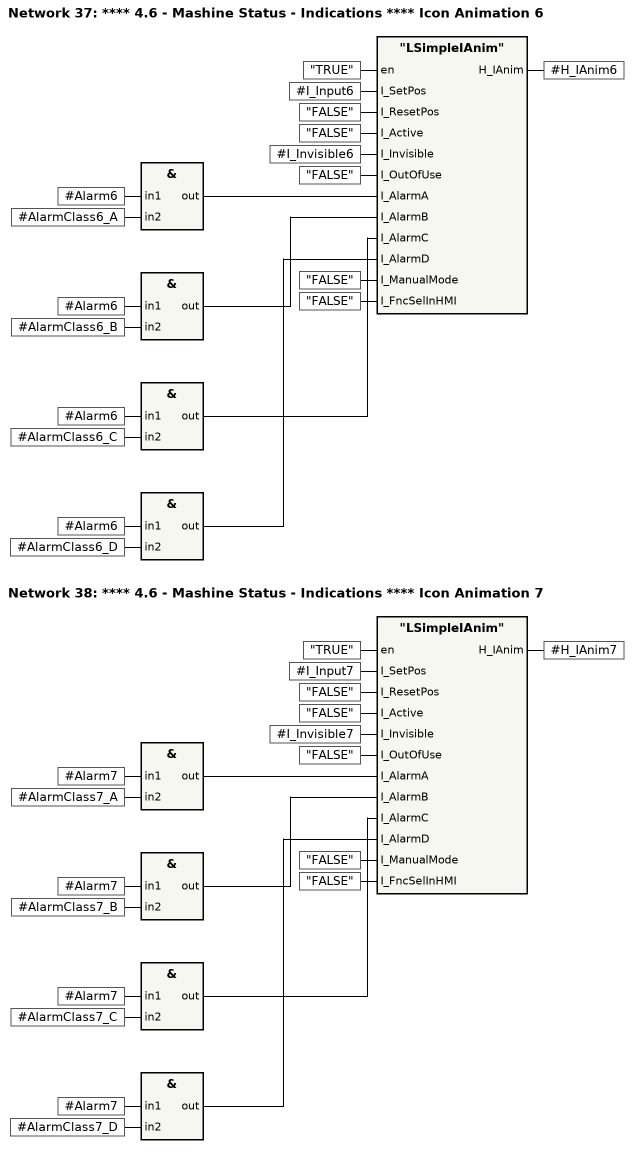
   IF "TRUE" THEN
       "LSimpleIAnim"(I_SetPos := #I_Input6,
                      I_ResetPos := "FALSE",
                      I_Active := "FALSE",
                      I_Invisible := #I_Invisible6,
                      I_OutOfUse := "FALSE",
                      I_AlarmA := #Alarm6 AND #AlarmClass6_A,
                      I_AlarmB := #Alarm6 AND #AlarmClass6_B,
                      I_AlarmC := #Alarm6 AND #AlarmClass6_C,
                      I_AlarmD := #Alarm6 AND #AlarmClass6_D,
                      I_ManualMode := "FALSE",
                      I_FncSelInHMI := "FALSE",
                      H_IAnim => #H_IAnim6);
   END_IF;
END_REGION

REGION Network 38: **** 4.6 - Mashine Status - Indications **** Icon Animation 7
   // Icon Animation 7
   IF "TRUE" THEN
       "LSimpleIAnim"(I_SetPos := #I_Input7,
                      I_ResetPos := "FALSE",
                      I_Active := "FALSE",
                      I_Invisible := #I_Invisible7,
                      I_OutOfUse := "FALSE",
                      I_AlarmA := #Alarm7 AND #AlarmClass7_A,
                      I_AlarmB := #Alarm7 AND #AlarmClass7_B,
                      I_AlarmC := #Alarm7 AND #AlarmClass7_C,
                      I_AlarmD := #Alarm7 AND #AlarmClass7_D,
                      I_ManualMode := "FALSE",
                      I_FncSelInHMI := "FALSE",
                      H_IAnim => #H_IAnim7);
   END_IF;
END_REGION

REGION Network 39: **** 4.6 - Mashine Status - Indications **** Icon Animation 8
   // Icon Animation 8
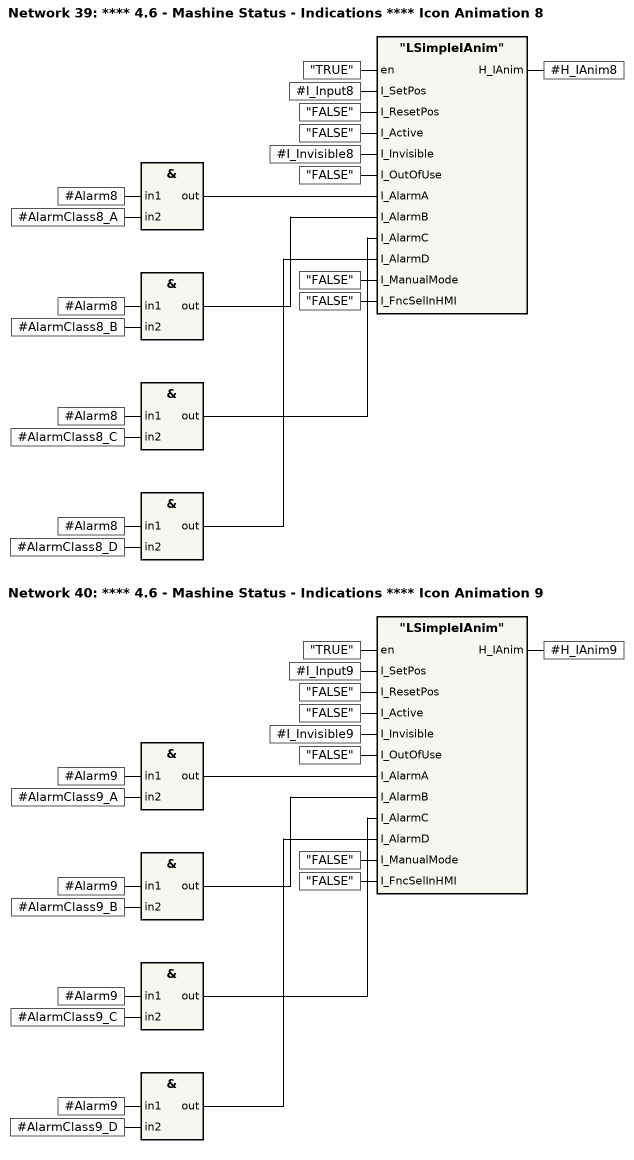
   IF "TRUE" THEN
       "LSimpleIAnim"(I_SetPos := #I_Input8,
                      I_ResetPos := "FALSE",
                      I_Active := "FALSE",
                      I_Invisible := #I_Invisible8,
                      I_OutOfUse := "FALSE",
                      I_AlarmA := #Alarm8 AND #AlarmClass8_A,
                      I_AlarmB := #Alarm8 AND #AlarmClass8_B,
                      I_AlarmC := #Alarm8 AND #AlarmClass8_C,
                      I_AlarmD := #Alarm8 AND #AlarmClass8_D,
                      I_ManualMode := "FALSE",
                      I_FncSelInHMI := "FALSE",
                      H_IAnim => #H_IAnim8);
   END_IF;
END_REGION

REGION Network 40: **** 4.6 - Mashine Status - Indications **** Icon Animation 9
   // Icon Animation 9
   IF "TRUE" THEN
       "LSimpleIAnim"(I_SetPos := #I_Input9,
                      I_ResetPos := "FALSE",
                      I_Active := "FALSE",
                      I_Invisible := #I_Invisible9,
                      I_OutOfUse := "FALSE",
                      I_AlarmA := #Alarm9 AND #AlarmClass9_A,
                      I_AlarmB := #Alarm9 AND #AlarmClass9_B,
                      I_AlarmC := #Alarm9 AND #AlarmClass9_C,
                      I_AlarmD := #Alarm9 AND #AlarmClass9_D,
                      I_ManualMode := "FALSE",
                      I_FncSelInHMI := "FALSE",
                      H_IAnim => #H_IAnim9);
   END_IF;
END_REGION

REGION Network 41: **** 4.6 - Mashine Status - Indications **** Icon Animation 10
   // Icon Animation 10
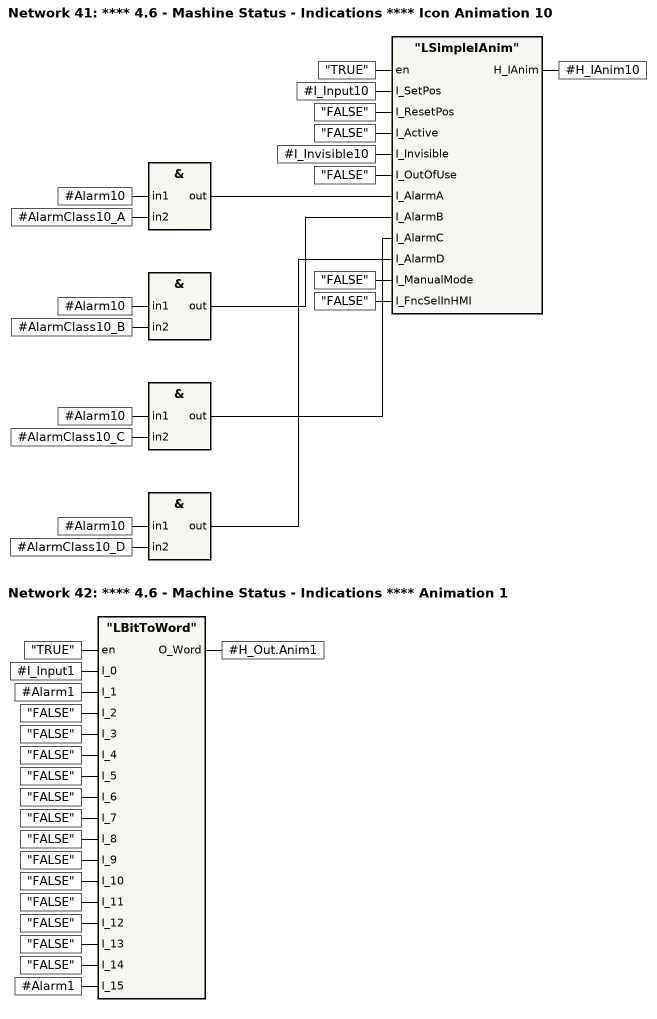
   IF "TRUE" THEN
       "LSimpleIAnim"(I_SetPos := #I_Input10,
                      I_ResetPos := "FALSE",
                      I_Active := "FALSE",
                      I_Invisible := #I_Invisible10,
                      I_OutOfUse := "FALSE",
                      I_AlarmA := #Alarm10 AND #AlarmClass10_A,
                      I_AlarmB := #Alarm10 AND #AlarmClass10_B,
                      I_AlarmC := #Alarm10 AND #AlarmClass10_C,
                      I_AlarmD := #Alarm10 AND #AlarmClass10_D,
                      I_ManualMode := "FALSE",
                      I_FncSelInHMI := "FALSE",
                      H_IAnim => #H_IAnim10);
   END_IF;
END_REGION

REGION Network 42: **** 4.6 - Machine Status - Indications **** Animation 1
   // Animation 1
   IF "TRUE" THEN
       "LBitToWord"(I_0 := #I_Input1,
                    I_1 := #Alarm1,
                    I_2 := "FALSE",
                    I_3 := "FALSE",
                    I_4 := "FALSE",
                    I_5 := "FALSE",
                    I_6 := "FALSE",
                    I_7 := "FALSE",
                    I_8 := "FALSE",
                    I_9 := "FALSE",
                    I_10 := "FALSE",
                    I_11 := "FALSE",
                    I_12 := "FALSE",
                    I_13 := "FALSE",
                    I_14 := "FALSE",
                    I_15 := #Alarm1,
                    O_Word => #H_Out.Anim1);
   END_IF;
END_REGION

REGION Network 43: **** 4.6 - Machine Status - Indications **** Animation 2
   // Animation 2
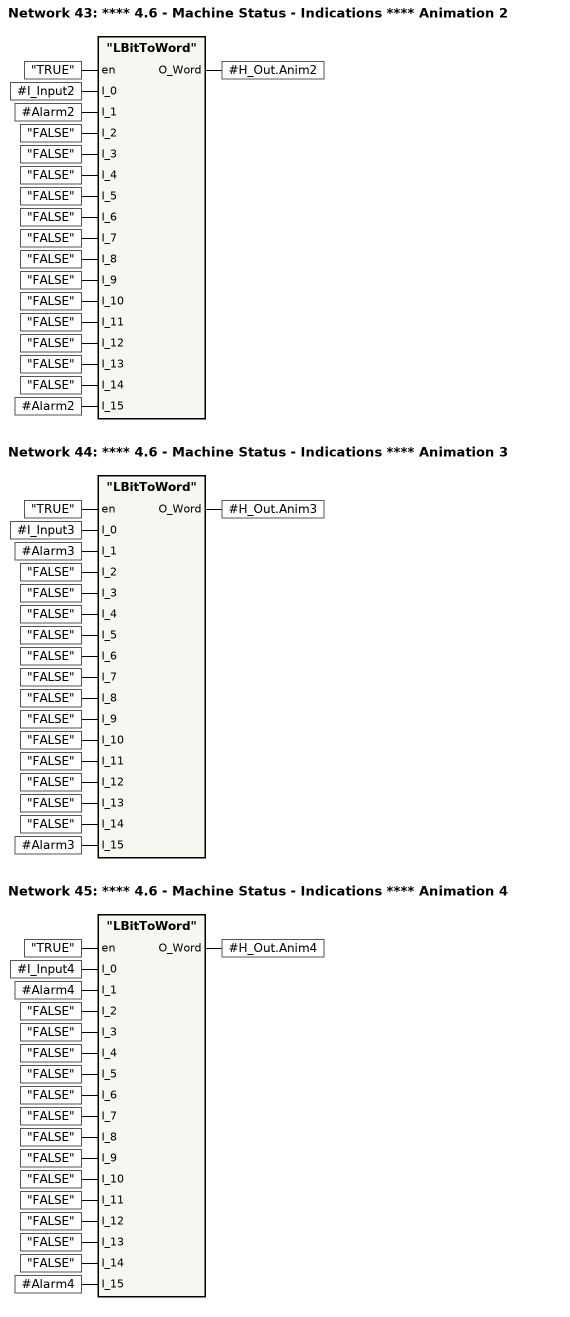
   IF "TRUE" THEN
       "LBitToWord"(I_0 := #I_Input2,
                    I_1 := #Alarm2,
                    I_2 := "FALSE",
                    I_3 := "FALSE",
                    I_4 := "FALSE",
                    I_5 := "FALSE",
                    I_6 := "FALSE",
                    I_7 := "FALSE",
                    I_8 := "FALSE",
                    I_9 := "FALSE",
                    I_10 := "FALSE",
                    I_11 := "FALSE",
                    I_12 := "FALSE",
                    I_13 := "FALSE",
                    I_14 := "FALSE",
                    I_15 := #Alarm2,
                    O_Word => #H_Out.Anim2);
   END_IF;
END_REGION

REGION Network 44: **** 4.6 - Machine Status - Indications **** Animation 3
   // Animation 3
   IF "TRUE" THEN
       "LBitToWord"(I_0 := #I_Input3,
                    I_1 := #Alarm3,
                    I_2 := "FALSE",
                    I_3 := "FALSE",
                    I_4 := "FALSE",
                    I_5 := "FALSE",
                    I_6 := "FALSE",
                    I_7 := "FALSE",
                    I_8 := "FALSE",
                    I_9 := "FALSE",
                    I_10 := "FALSE",
                    I_11 := "FALSE",
                    I_12 := "FALSE",
                    I_13 := "FALSE",
                    I_14 := "FALSE",
                    I_15 := #Alarm3,
                    O_Word => #H_Out.Anim3);
   END_IF;
END_REGION

REGION Network 45: **** 4.6 - Machine Status - Indications **** Animation 4
   // Animation 4
   IF "TRUE" THEN
       "LBitToWord"(I_0 := #I_Input4,
                    I_1 := #Alarm4,
                    I_2 := "FALSE",
                    I_3 := "FALSE",
                    I_4 := "FALSE",
                    I_5 := "FALSE",
                    I_6 := "FALSE",
                    I_7 := "FALSE",
                    I_8 := "FALSE",
                    I_9 := "FALSE",
                    I_10 := "FALSE",
                    I_11 := "FALSE",
                    I_12 := "FALSE",
                    I_13 := "FALSE",
                    I_14 := "FALSE",
                    I_15 := #Alarm4,
                    O_Word => #H_Out.Anim4);
   END_IF;
END_REGION

REGION Network 46: **** 4.6 - Machine Status - Indications **** Animation 5
   // Animation 5
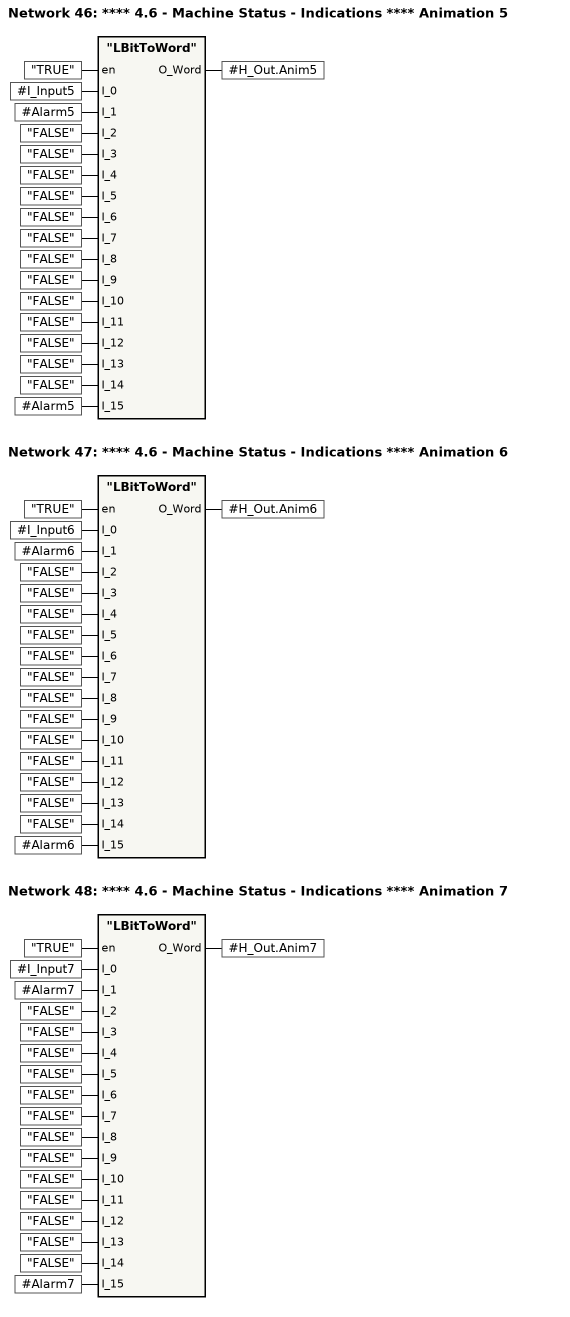
   IF "TRUE" THEN
       "LBitToWord"(I_0 := #I_Input5,
                    I_1 := #Alarm5,
                    I_2 := "FALSE",
                    I_3 := "FALSE",
                    I_4 := "FALSE",
                    I_5 := "FALSE",
                    I_6 := "FALSE",
                    I_7 := "FALSE",
                    I_8 := "FALSE",
                    I_9 := "FALSE",
                    I_10 := "FALSE",
                    I_11 := "FALSE",
                    I_12 := "FALSE",
                    I_13 := "FALSE",
                    I_14 := "FALSE",
                    I_15 := #Alarm5,
                    O_Word => #H_Out.Anim5);
   END_IF;
END_REGION

REGION Network 47: **** 4.6 - Machine Status - Indications **** Animation 6
   // Animation 6
   IF "TRUE" THEN
       "LBitToWord"(I_0 := #I_Input6,
                    I_1 := #Alarm6,
                    I_2 := "FALSE",
                    I_3 := "FALSE",
                    I_4 := "FALSE",
                    I_5 := "FALSE",
                    I_6 := "FALSE",
                    I_7 := "FALSE",
                    I_8 := "FALSE",
                    I_9 := "FALSE",
                    I_10 := "FALSE",
                    I_11 := "FALSE",
                    I_12 := "FALSE",
                    I_13 := "FALSE",
                    I_14 := "FALSE",
                    I_15 := #Alarm6,
                    O_Word => #H_Out.Anim6);
   END_IF;
END_REGION

REGION Network 48: **** 4.6 - Machine Status - Indications **** Animation 7
   // Animation 7
   IF "TRUE" THEN
       "LBitToWord"(I_0 := #I_Input7,
                    I_1 := #Alarm7,
                    I_2 := "FALSE",
                    I_3 := "FALSE",
                    I_4 := "FALSE",
                    I_5 := "FALSE",
                    I_6 := "FALSE",
                    I_7 := "FALSE",
                    I_8 := "FALSE",
                    I_9 := "FALSE",
                    I_10 := "FALSE",
                    I_11 := "FALSE",
                    I_12 := "FALSE",
                    I_13 := "FALSE",
                    I_14 := "FALSE",
                    I_15 := #Alarm7,
                    O_Word => #H_Out.Anim7);
   END_IF;
END_REGION

REGION Network 49: **** 4.6 - Machine Status - Indications **** Animation 8
   // Animation 8
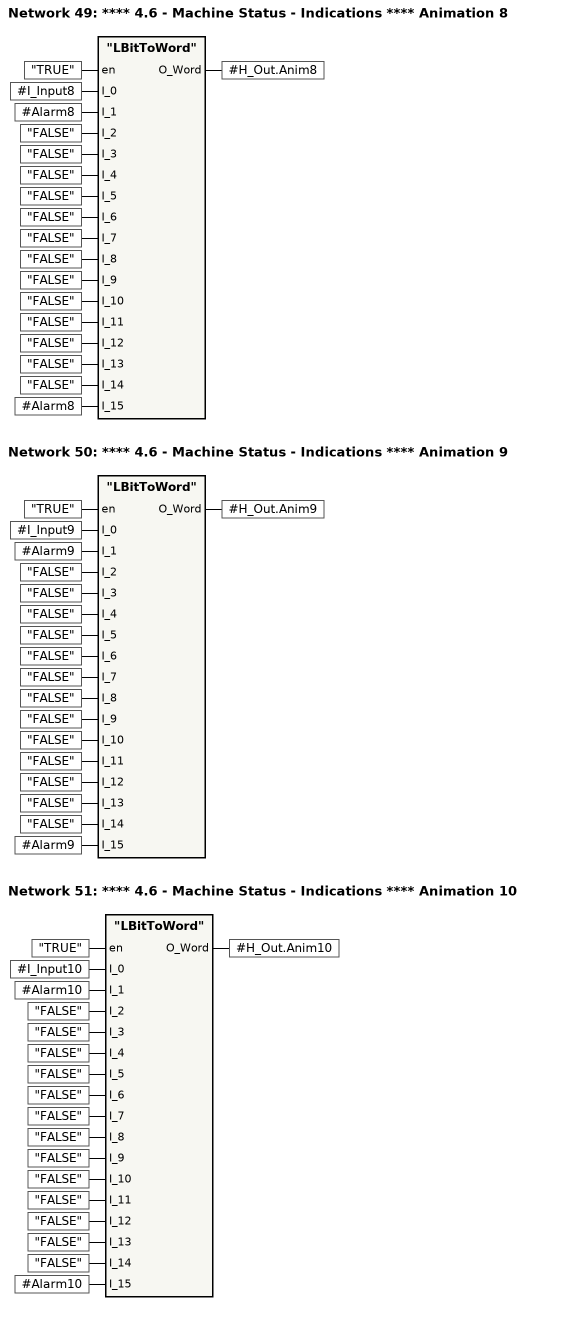
   IF "TRUE" THEN
       "LBitToWord"(I_0 := #I_Input8,
                    I_1 := #Alarm8,
                    I_2 := "FALSE",
                    I_3 := "FALSE",
                    I_4 := "FALSE",
                    I_5 := "FALSE",
                    I_6 := "FALSE",
                    I_7 := "FALSE",
                    I_8 := "FALSE",
                    I_9 := "FALSE",
                    I_10 := "FALSE",
                    I_11 := "FALSE",
                    I_12 := "FALSE",
                    I_13 := "FALSE",
                    I_14 := "FALSE",
                    I_15 := #Alarm8,
                    O_Word => #H_Out.Anim8);
   END_IF;
END_REGION

REGION Network 50: **** 4.6 - Machine Status - Indications **** Animation 9
   // Animation 9
   IF "TRUE" THEN
       "LBitToWord"(I_0 := #I_Input9,
                    I_1 := #Alarm9,
                    I_2 := "FALSE",
                    I_3 := "FALSE",
                    I_4 := "FALSE",
                    I_5 := "FALSE",
                    I_6 := "FALSE",
                    I_7 := "FALSE",
                    I_8 := "FALSE",
                    I_9 := "FALSE",
                    I_10 := "FALSE",
                    I_11 := "FALSE",
                    I_12 := "FALSE",
                    I_13 := "FALSE",
                    I_14 := "FALSE",
                    I_15 := #Alarm9,
                    O_Word => #H_Out.Anim9);
   END_IF;
END_REGION

REGION Network 51: **** 4.6 - Machine Status - Indications **** Animation 10
   // Animation 10
   IF "TRUE" THEN
       "LBitToWord"(I_0 := #I_Input10,
                    I_1 := #Alarm10,
                    I_2 := "FALSE",
                    I_3 := "FALSE",
                    I_4 := "FALSE",
                    I_5 := "FALSE",
                    I_6 := "FALSE",
                    I_7 := "FALSE",
                    I_8 := "FALSE",
                    I_9 := "FALSE",
                    I_10 := "FALSE",
                    I_11 := "FALSE",
                    I_12 := "FALSE",
                    I_13 := "FALSE",
                    I_14 := "FALSE",
                    I_15 := #Alarm10,
                    O_Word => #H_Out.Anim10);
   END_IF;
END_REGION

REGION Network 52: **** 4.6 - Machine status - Indications **** Animation DB number
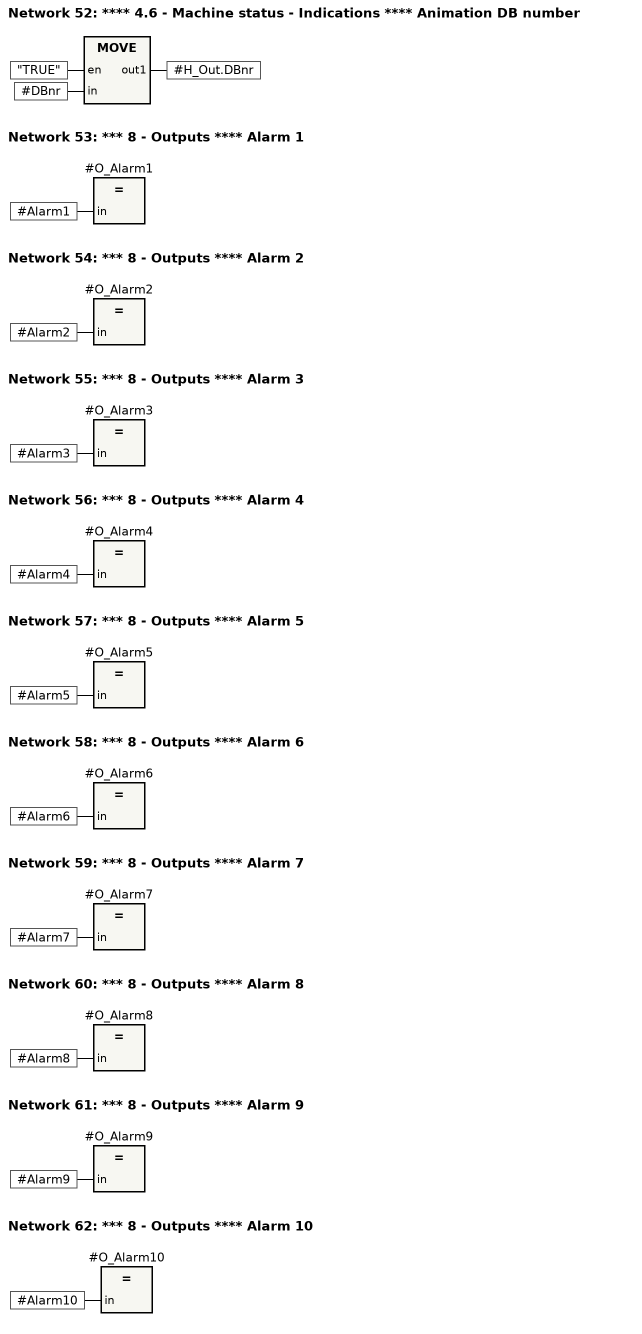
   IF "TRUE" THEN #H_Out.DBnr := #DBnr; END_IF;
END_REGION

REGION Network 53: *** 8 - Outputs **** Alarm 1
   // Output of the Alarm 1
   #O_Alarm1 := #Alarm1;
END_REGION

REGION Network 54: *** 8 - Outputs **** Alarm 2
   // Output of the Alarm 2
   #O_Alarm2 := #Alarm2;
END_REGION

REGION Network 55: *** 8 - Outputs **** Alarm 3
   // Output of the Alarm 3
   #O_Alarm3 := #Alarm3;
END_REGION

REGION Network 56: *** 8 - Outputs **** Alarm 4
   // Output of the Alarm 4
   #O_Alarm4 := #Alarm4;
END_REGION

REGION Network 57: *** 8 - Outputs **** Alarm 5
   // Output of the Alarm 5
   #O_Alarm5 := #Alarm5;
END_REGION

REGION Network 58: *** 8 - Outputs **** Alarm 6
   // Output of the Alarm 6
   #O_Alarm6 := #Alarm6;
END_REGION

REGION Network 59: *** 8 - Outputs **** Alarm 7
   // Output of the Alarm 7
   #O_Alarm7 := #Alarm7;
END_REGION

REGION Network 60: *** 8 - Outputs **** Alarm 8
   // Output of the Alarm 8
   #O_Alarm8 := #Alarm8;
END_REGION

REGION Network 61: *** 8 - Outputs **** Alarm 9
   // Output of the Alarm 9
   #O_Alarm9 := #Alarm9;
END_REGION

REGION Network 62: *** 8 - Outputs **** Alarm 10
   // Output of the Alarm 10
   #O_Alarm10 := #Alarm10;
END_REGION

REGION Network 63: **** 8 - Outputs **** Alarm AB Condition
   // Alarm AB condition
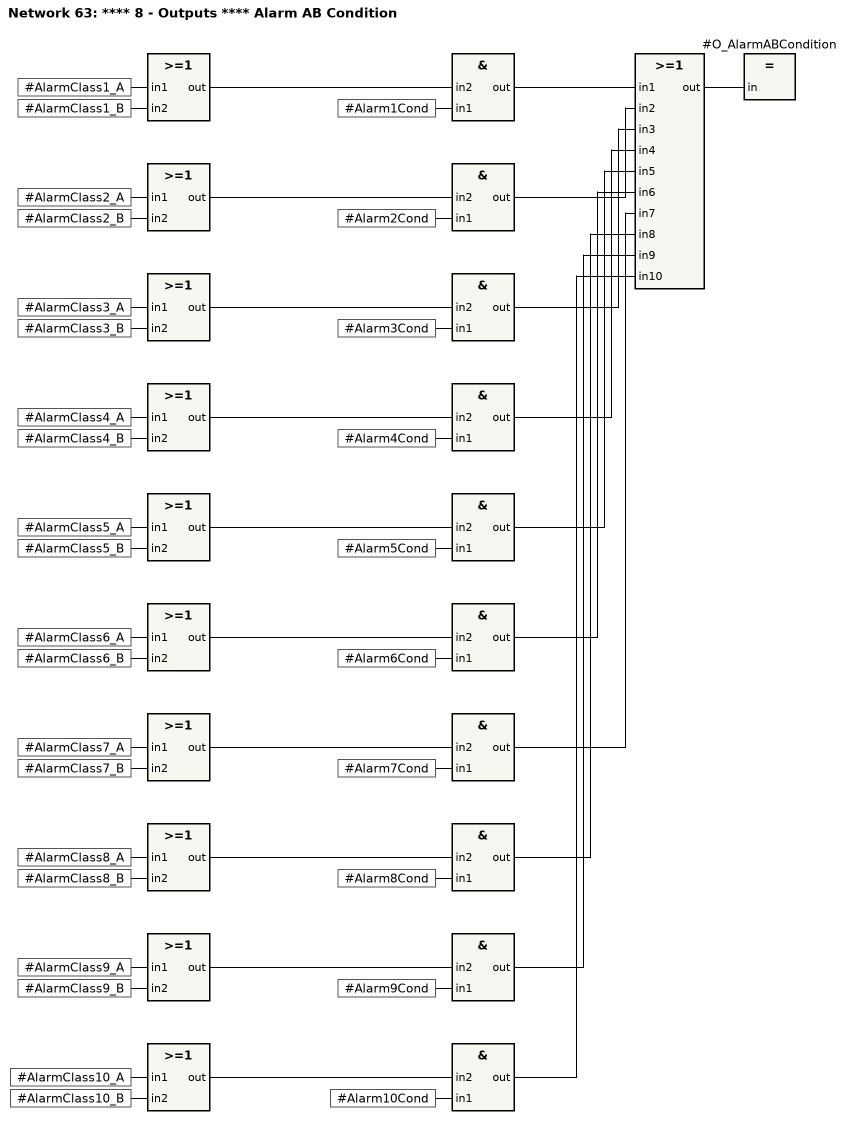
   #O_AlarmABCondition := ((#AlarmClass1_A OR #AlarmClass1_B) AND #Alarm1Cond) OR ((#AlarmClass2_A OR #AlarmClass2_B) AND #Alarm2Cond) OR ((#AlarmClass3_A OR #AlarmClass3_B) AND #Alarm3Cond) OR ((#AlarmClass4_A OR #AlarmClass4_B) AND #Alarm4Cond) OR ((#AlarmClass5_A OR #AlarmClass5_B) AND #Alarm5Cond) OR ((#AlarmClass6_A OR #AlarmClass6_B) AND #Alarm6Cond) OR ((#AlarmClass7_A OR #AlarmClass7_B) AND #Alarm7Cond) OR ((#AlarmClass8_A OR #AlarmClass8_B) AND #Alarm8Cond) OR ((#AlarmClass9_A OR #AlarmClass9_B) AND #Alarm9Cond) OR ((#AlarmClass10_A OR #AlarmClass10_B) AND #Alarm10Cond);
END_REGION
END_FUNCTION_BLOCK

FUNCTION_BLOCK "LLoccBoxAlarm"   // FB1411, FBD
TITLE = LLoccBoxAlarm
{ S7_Optimized_Access := 'FALSE' }
AUTHOR : VCG
FAMILY : AlarmHnd
NAME : SpcGB
VERSION : 1.0
// ================================================================================
// This module is used for installations with Locc-Box type 7-6410.
// It create alarms and warning in function of configuration and status from the 
// Box.
// It Send Mode byte to the Box in function of Pop-up and external commands
// ================================================================================
// C_AlarmOrWarning
// Bit0: C_LevelOFF (Bit ON=Warning ; OFF=Alarm)
// Bit1: C_LevelBlown (Bit ON=Warning ; OFF=Alarm)
// Bit2: C_LevelExtOFF (Bit ON=Warning ; OFF=Alarm)
// Bit3: C_LevelCurrentLimit (Bit ON=Warning ; OFF=Alarm)
// Bit4: C_LevelUndVolt (Bit ON=Warning ; OFF=Alarm)
// Bit5: C_LevelShortCirc (Bit ON=Warning ; OFF=Alarm)
// Bit6: C_LevelSystError (Bit ON=Warning ; OFF=Alarm)
// Bit7: C_LevelSpareBit7
// Bit8: C_LevelSpareBit8
// Bit9: C_LevelSpareBit9
// Bit10:C_LevelSpareBit10
// Bit11:C_LevelSpareBit11
// Bit12:C_LevelSpareBit12
// Bit13:C_LevelSpareBit13
// Bit14:C_LevelSpareBit14
// Bit15:C_LevelSpareBit15
// ================================================================================
// H_HMICmd
// Bit0: HMICmdSwitchON (Bit PosEdge = Request ON)
// Bit1: HMICmdSwitchOFF (Bit PosEdge = Request OFF)
// Bit2: HMICmdResetOFF (Bit PosEdge = Reset OFF)
// Bit3: HMICmdResetExtOFF (Bit PosEdge = Reset ExtOFF)
// Bit4: HMICmdResetCurrentLimit(Bit PosEdge = Reset CurrentLimit)
// Bit5: HMICmdResetUndVolt(Bit PosEdge = Reset UndVolt)
// Bit6: HMICmdResetShortCirc(Bit PosEdge = Reset ShortCirc)
// Bit7: HMICmdResetSystError(Bit PosEdge = Reset SystError)
// Bit8: HMICmdSpareBit8
// Bit9: HMICmdSpareBit9
// Bit10:HMICmdSpareBit10
// Bit11:HMICmdSpareBit11
// Bit12:HMICmdSpareBit12
// Bit13:HMICmdSpareBit13
// Bit14:HMICmdSpareBit14
// Bit15:HMICmdSpareBit15
// ================================================================================
// C_LocalOrRemoteReset
// Bit0: C_LocalResetOFF (Bit ON=LocalResetOnly ; OFF=RemoteResetPossible)
// Bit1: C_LocalResetBlown (Bit ON=LocalResetOnly ; OFF=RemoteResetPossible)
// Bit2: C_LocalResetExtOFF (Bit ON=LocalResetOnly ; OFF=RemoteResetPossible)
// Bit3: C_LocalResetCurrentLimit (Bit ON=LocalResetOnly ; OFF=RemoteResetPossible)
// Bit4: C_LocalResetUndVolt (Bit ON=LocalResetOnly ; OFF=RemoteResetPossible)
// Bit5: C_LocalResetShortCirc (Bit ON=LocalResetOnly ; OFF=RemoteResetPossible)
// Bit6: C_LocalResetSystError (Bit ON=LocalResetOnly ; OFF=RemoteResetPossible)
// Bit7: C_LocalResetBit7
// Bit8: C_LocalResetBit8
// Bit9: C_LocalResetBit9
// Bit10:C_LocalResetBit10
// Bit11:C_LocalResetBit11
// Bit12:C_LocalResetBit12
// Bit13:C_LocalResetBit13
// Bit14:C_LocalResetBit14
// Bit15:C_LocalResetBit15
// 
// Updated to make fuse resetable from WinCC (Through HMI cmd)
// stored: AutoNumber false, IsIECCheckEnabled false, SetENOAutomatically False, UDAEnableTagReadback false
   VAR_INPUT
      I_IBState { ExternalAccessible := 'False'; ExternalVisible := 'False'; ExternalWritable := 'False'} : Byte;   // Input Byte state from Locc-Box
      I_HWSubModule { ExternalAccessible := 'False'; ExternalVisible := 'False'; ExternalWritable := 'False'} : HW_SUBMODULE;   // Connection with Hardware Sub Module
      I_RotarySwitchCurrent { ExternalAccessible := 'False'; ExternalVisible := 'False'; ExternalWritable := 'False'} : Int;   // Setting current -> rotary switch on the fuse
      I_RotarySwitchCurve { ExternalAccessible := 'False'; ExternalVisible := 'False'; ExternalWritable := 'False'} : Int;   // Setting curve -> rotary switch on the fuse
      I_AlarmClass { ExternalAccessible := 'False'; ExternalVisible := 'False'; ExternalWritable := 'False'} : Char;   // Alarm class -> A - B or C / Alarm class -> A - B - C or D
      I_EnableAlarm { ExternalAccessible := 'False'; ExternalVisible := 'False'; ExternalWritable := 'False'} : Bool := TRUE;   // Enable alarm from upper level
      I_AlarmResetPB { ExternalAccessible := 'False'; ExternalVisible := 'False'; ExternalWritable := 'False'} : Bool;   // Alarm reset pushbutton is activated
      C_AlarmOrWarning { ExternalAccessible := 'False'; ExternalVisible := 'False'; ExternalWritable := 'False'} : Word;   // Used to define if for this installation a status is alarm or warning
      C_LocalOrRemoteReset { ExternalAccessible := 'False'; ExternalVisible := 'False'; ExternalWritable := 'False'} : Word;   // Used to define if for this installation an error is local or remote reset
   END_VAR
   VAR_OUTPUT
      O_OBMode { ExternalAccessible := 'False'; ExternalVisible := 'False'; ExternalWritable := 'False'} : Byte;   // Output Byte Mode to Locc-Box
      O_Alarm { ExternalAccessible := 'False'; ExternalVisible := 'False'; ExternalWritable := 'False'} : Bool;   // Alarm state from the Locc-Box (Alarm list done inside)
      O_Warning { ExternalAccessible := 'False'; ExternalVisible := 'False'; ExternalWritable := 'False'} : Bool;   // Warning state from the Locc-Box (Alarm list done inside)
      O_AlarmABCondition { ExternalAccessible := 'False'; ExternalVisible := 'False'; ExternalWritable := 'False'} : Bool;   // Alarm AB condition
      H_IAnim { ExternalAccessible := 'False'; ExternalVisible := 'False'; ExternalWritable := 'False'} : Word;   // HMI Animation color of the icon
      H_AlarmWord { ExternalAccessible := 'False'; ExternalVisible := 'False'; ExternalWritable := 'False'} : DWord;   // Alarm Word
   END_VAR
   VAR_IN_OUT
      IO_GlobalSignals : Struct   // Global signals between all the FB's
         Busy : Bool;   // Busy with GET the info from one of the fuses
         DBnrFromPopup : Int;   // The return DB number from the pop-up that is open
      END_STRUCT;
   END_VAR
   VAR DB_SPECIFIC
      AA_AlarmOFF { ExternalAccessible := 'False'; ExternalVisible := 'False'; ExternalWritable := 'False'} : Bool;   // Fuse Locc-Box is switch OFF / Extra Info Locc-Box Fuse -> Is switch OFF
      AA_AlarmBlown { ExternalAccessible := 'False'; ExternalVisible := 'False'; ExternalWritable := 'False'} : Bool;   // Fuse Locc-Box Blown Alarm / Extra Info Locc-Box Fuse -> Blown Alarm
      AA_AlarmExtOFF { ExternalAccessible := 'False'; ExternalVisible := 'False'; ExternalWritable := 'False'} : Bool;   // Fuse Locc-Box External OFF Alarm / Extra Info Locc-Box Fuse -> External OFF Alarm
      AA_AlarmCurrentLimit { ExternalAccessible := 'False'; ExternalVisible := 'False'; ExternalWritable := 'False'} : Bool;   // Fuse Locc-Box Current Limit Alarm / Extra Info Locc-Box Fuse -> Current Limit Alarm
      AA_AlarmUndVolt { ExternalAccessible := 'False'; ExternalVisible := 'False'; ExternalWritable := 'False'} : Bool;   // Fuse Locc-Box Under Voltage Alarm / Extra Info Locc-Box Fuse -> Under Voltage Alarm
      AA_AlarmShortCirc { ExternalAccessible := 'False'; ExternalVisible := 'False'; ExternalWritable := 'False'} : Bool;   // Fuse Locc-Box Short circuit Alarm / Extra Info Locc-Box Fuse -> Short circuit Alarm
      AA_AlarmSystError { ExternalAccessible := 'False'; ExternalVisible := 'False'; ExternalWritable := 'False'} : Bool;   // Fuse Locc-Box System error Alarm / Extra Info Locc-Box Fuse -> System error Alarm
      AB_AlarmOFF { ExternalAccessible := 'False'; ExternalVisible := 'False'; ExternalWritable := 'False'} : Bool;   // Fuse Locc-Box is switch OFF / Extra Info Locc-Box Fuse -> Is switch OFF
      AB_AlarmBlown { ExternalAccessible := 'False'; ExternalVisible := 'False'; ExternalWritable := 'False'} : Bool;   // Fuse Locc-Box Blown Alarm / Extra Info Locc-Box Fuse -> Blown Alarm
      AB_AlarmExtOFF { ExternalAccessible := 'False'; ExternalVisible := 'False'; ExternalWritable := 'False'} : Bool;   // Fuse Locc-Box External OFF Alarm / Extra Info Locc-Box Fuse -> External OFF Alarm
      AB_AlarmCurrentLimit { ExternalAccessible := 'False'; ExternalVisible := 'False'; ExternalWritable := 'False'} : Bool;   // Fuse Locc-Box Current Limit Alarm / Extra Info Locc-Box Fuse -> Current Limit Alarm
      AB_AlarmUndVolt { ExternalAccessible := 'False'; ExternalVisible := 'False'; ExternalWritable := 'False'} : Bool;   // Fuse Locc-Box Under Voltage Alarm / Extra Info Locc-Box Fuse -> Under Voltage Alarm
      AB_AlarmShortCirc { ExternalAccessible := 'False'; ExternalVisible := 'False'; ExternalWritable := 'False'} : Bool;   // Fuse Locc-Box Short circuit Alarm / Extra Info Locc-Box Fuse -> Short circuit Alarm
      AB_AlarmSystError { ExternalAccessible := 'False'; ExternalVisible := 'False'; ExternalWritable := 'False'} : Bool;   // Fuse Locc-Box System error Alarm / Extra Info Locc-Box Fuse -> System error Alarm
      AC_AlarmOFF { ExternalAccessible := 'False'; ExternalVisible := 'False'; ExternalWritable := 'False'} : Bool;   // Fuse Locc-Box is switch OFF / Extra Info Locc-Box Fuse -> Is switch OFF
      AC_AlarmBlown { ExternalAccessible := 'False'; ExternalVisible := 'False'; ExternalWritable := 'False'} : Bool;   // Fuse Locc-Box Blown Alarm / Extra Info Locc-Box Fuse -> Blown Alarm
      AC_AlarmExtOFF { ExternalAccessible := 'False'; ExternalVisible := 'False'; ExternalWritable := 'False'} : Bool;   // Fuse Locc-Box External OFF Alarm / Extra Info Locc-Box Fuse -> External OFF Alarm
      AC_AlarmCurrentLimit { ExternalAccessible := 'False'; ExternalVisible := 'False'; ExternalWritable := 'False'} : Bool;   // Fuse Locc-Box Current Limit Alarm / Extra Info Locc-Box Fuse -> Current Limit Alarm
      AC_AlarmUndVolt { ExternalAccessible := 'False'; ExternalVisible := 'False'; ExternalWritable := 'False'} : Bool;   // Fuse Locc-Box Under Voltage Alarm / Extra Info Locc-Box Fuse -> Under Voltage Alarm
      AC_AlarmShortCirc { ExternalAccessible := 'False'; ExternalVisible := 'False'; ExternalWritable := 'False'} : Bool;   // Fuse Locc-Box Short circuit Alarm / Extra Info Locc-Box Fuse -> Short circuit Alarm
      AC_AlarmSystError { ExternalAccessible := 'False'; ExternalVisible := 'False'; ExternalWritable := 'False'} : Bool;   // Fuse Locc-Box System error Alarm / Extra Info Locc-Box Fuse -> System error Alarm
      AD_WarningOFF { ExternalAccessible := 'False'; ExternalVisible := 'False'; ExternalWritable := 'False'} : Bool;   // Fuse Locc-Box OFF Warning / Extra Info Locc-Box Fuse -> OFF Warning
      AD_WarningBlown { ExternalAccessible := 'False'; ExternalVisible := 'False'; ExternalWritable := 'False'} : Bool;   // Fuse Locc-Box Blown Warning / Extra Info Locc-Box Fuse -> Blown Warning
      AD_WarningExtOFF { ExternalAccessible := 'False'; ExternalVisible := 'False'; ExternalWritable := 'False'} : Bool;   // Fuse Locc-Box External OFF Warning / Extra Info Locc-Box Fuse -> External OFF Warning
      AD_WarningCurrentLimit { ExternalAccessible := 'False'; ExternalVisible := 'False'; ExternalWritable := 'False'} : Bool;   // Fuse Locc-Box Current Limit Warning / Extra Info Locc-Box Fuse -> Current Limit Warning
      AD_WarningUndVolt { ExternalAccessible := 'False'; ExternalVisible := 'False'; ExternalWritable := 'False'} : Bool;   // Fuse Locc-Box Under Voltage Warning / Extra Info Locc-Box Fuse -> Under Voltage Warning
      AD_WarningShortCirc { ExternalAccessible := 'False'; ExternalVisible := 'False'; ExternalWritable := 'False'} : Bool;   // Fuse Locc-Box Short circuit Warning / Extra Info Locc-Box Fuse -> Short circuit Warning
      AD_WarningSystError { ExternalAccessible := 'False'; ExternalVisible := 'False'; ExternalWritable := 'False'} : Bool;   // Fuse Locc-Box System error Warning / Extra Info Locc-Box Fuse -> System error Warning
      AD_RotarySwitchCurrent { ExternalAccessible := 'False'; ExternalVisible := 'False'; ExternalWritable := 'False'} : Bool;   // Rotary switch on the fuse is changed for the current / Extra Info Locc-Box Fuse -> Rotary switch on the fuse is changed for the current
      AD_RotarySwitchCurve { ExternalAccessible := 'False'; ExternalVisible := 'False'; ExternalWritable := 'False'} : Bool;   // Rotary switch on the fuse is changed for the curve / Extra Info Locc-Box Fuse -> Rotary switch on the fuse is changed for the curve
      H_HMICmd : Word;   // HMI Command from Pop-Up
      H_Out : Struct   // HMI
         Anim : Word;   // HMI Animation Word
         Anim2 : Word;   // HMI Animation Word
         Anim3 : Word;   // HMI Animation Word
         InputVoltage : Real;   // HMI Input Voltage
         OutputVoltage : Real;   // HMI Output Voltage
         CurrentSetp : Int;   // HMI Current setpoint
         ActCurrent : Real;   // HMI Actual Current
         Curve : Int;   // HMI Curve type
         CurveSTRING : String[25];   // HMI Curve type
         DBnr : Int;   // HMI Animation DB number
      END_STRUCT;
      AlarmOFF { ExternalAccessible := 'False'; ExternalVisible := 'False'; ExternalWritable := 'False'} : Bool;   // Fuse Locc-Box is switch OFF / Fuse Locc-Box Is switch OFF
      AlarmBlown { ExternalAccessible := 'False'; ExternalVisible := 'False'; ExternalWritable := 'False'} : Bool;   // Fuse Locc-Box Blown Alarm
      AlarmExtOFF { ExternalAccessible := 'False'; ExternalVisible := 'False'; ExternalWritable := 'False'} : Bool;   // Fuse Locc-Box External OFF Alarm
      AlarmCurrentLimit { ExternalAccessible := 'False'; ExternalVisible := 'False'; ExternalWritable := 'False'} : Bool;   // Fuse Locc-Box Current Limit Alarm
      AlarmUndVolt { ExternalAccessible := 'False'; ExternalVisible := 'False'; ExternalWritable := 'False'} : Bool;   // Fuse Locc-Box Under Voltage Alarm
      AlarmShortCirc { ExternalAccessible := 'False'; ExternalVisible := 'False'; ExternalWritable := 'False'} : Bool;   // Fuse Locc-Box Short circuit Alarm
      AlarmSystError { ExternalAccessible := 'False'; ExternalVisible := 'False'; ExternalWritable := 'False'} : Bool;   // Fuse Locc-Box System error Alarm
      AlarmCondOFF { ExternalAccessible := 'False'; ExternalVisible := 'False'; ExternalWritable := 'False'} : Bool;   // Alarm condition
      AlarmCondBlown { ExternalAccessible := 'False'; ExternalVisible := 'False'; ExternalWritable := 'False'} : Bool;   // Alarm condition
      AlarmCondExtOFF { ExternalAccessible := 'False'; ExternalVisible := 'False'; ExternalWritable := 'False'} : Bool;   // Alarm condition
      AlarmCondCurrentLimit { ExternalAccessible := 'False'; ExternalVisible := 'False'; ExternalWritable := 'False'} : Bool;   // Alarm condition
      AlarmCondUndVolt { ExternalAccessible := 'False'; ExternalVisible := 'False'; ExternalWritable := 'False'} : Bool;   // Alarm condition
      AlarmCondShortCirc { ExternalAccessible := 'False'; ExternalVisible := 'False'; ExternalWritable := 'False'} : Bool;   // Alarm condition
      AlarmCondSystError { ExternalAccessible := 'False'; ExternalVisible := 'False'; ExternalWritable := 'False'} : Bool;   // Alarm condition
      Alarm { ExternalAccessible := 'False'; ExternalVisible := 'False'; ExternalWritable := 'False'} : Bool;   // Alarm
      Warning { ExternalAccessible := 'False'; ExternalVisible := 'False'; ExternalWritable := 'False'} : Bool;   // Warning
      AlarmClass_A { ExternalAccessible := 'False'; ExternalVisible := 'False'; ExternalWritable := 'False'} : Bool;   // The alarm is from alarm class A
      AlarmClass_B { ExternalAccessible := 'False'; ExternalVisible := 'False'; ExternalWritable := 'False'} : Bool;   // The alarm is from alarm class B
      AlarmClass_C { ExternalAccessible := 'False'; ExternalVisible := 'False'; ExternalWritable := 'False'} : Bool;   // The alarm is from alarm class C
      AlarmClass_D { ExternalAccessible := 'False'; ExternalVisible := 'False'; ExternalWritable := 'False'} : Bool;   // The alarm is from alarm class C / The alarm is from alarm class D
      C_LevelOFF { ExternalAccessible := 'False'; ExternalVisible := 'False'; ExternalWritable := 'False'} : Bool;   // Config alarm level
      C_LevelBlown { ExternalAccessible := 'False'; ExternalVisible := 'False'; ExternalWritable := 'False'} : Bool;   // Config alarm level
      C_LevelExtOFF { ExternalAccessible := 'False'; ExternalVisible := 'False'; ExternalWritable := 'False'} : Bool;   // Config alarm level
      C_LevelCurrentLimit { ExternalAccessible := 'False'; ExternalVisible := 'False'; ExternalWritable := 'False'} : Bool;   // Config alarm level
      C_LevelUndVolt { ExternalAccessible := 'False'; ExternalVisible := 'False'; ExternalWritable := 'False'} : Bool;   // Config alarm level
      C_LevelShortCirc { ExternalAccessible := 'False'; ExternalVisible := 'False'; ExternalWritable := 'False'} : Bool;   // Config alarm level
      C_LevelSystError { ExternalAccessible := 'False'; ExternalVisible := 'False'; ExternalWritable := 'False'} : Bool;   // Config alarm level
      C_LevelSpareBit7 { ExternalAccessible := 'False'; ExternalVisible := 'False'; ExternalWritable := 'False'} : Bool;   // Config alarm level
      C_LevelSpareBit8 { ExternalAccessible := 'False'; ExternalVisible := 'False'; ExternalWritable := 'False'} : Bool;   // Config alarm level
      C_LevelSpareBit9 { ExternalAccessible := 'False'; ExternalVisible := 'False'; ExternalWritable := 'False'} : Bool;   // Config alarm level
      C_LevelSpareBit10 { ExternalAccessible := 'False'; ExternalVisible := 'False'; ExternalWritable := 'False'} : Bool;   // Config alarm level
      C_LevelSpareBit11 { ExternalAccessible := 'False'; ExternalVisible := 'False'; ExternalWritable := 'False'} : Bool;   // Config alarm level
      C_LevelSpareBit12 { ExternalAccessible := 'False'; ExternalVisible := 'False'; ExternalWritable := 'False'} : Bool;   // Config alarm level
      C_LevelSpareBit13 { ExternalAccessible := 'False'; ExternalVisible := 'False'; ExternalWritable := 'False'} : Bool;   // Config alarm level
      C_LevelSpareBit14 { ExternalAccessible := 'False'; ExternalVisible := 'False'; ExternalWritable := 'False'} : Bool;   // Config alarm level
      C_LevelSpareBit15 { ExternalAccessible := 'False'; ExternalVisible := 'False'; ExternalWritable := 'False'} : Bool;   // Config alarm level
      HMICmdSwitchON { ExternalAccessible := 'False'; ExternalVisible := 'False'; ExternalWritable := 'False'} : Bool;   // HMICmd
      HMICmdSwitchOFF { ExternalAccessible := 'False'; ExternalVisible := 'False'; ExternalWritable := 'False'} : Bool;   // HMICmd
      HMICmdResetOFF { ExternalAccessible := 'False'; ExternalVisible := 'False'; ExternalWritable := 'False'} : Bool;   // HMICmd
      HMICmdResetBlown { ExternalAccessible := 'False'; ExternalVisible := 'False'; ExternalWritable := 'False'} : Bool;   // HMICmd
      HMICmdResetExtOFF { ExternalAccessible := 'False'; ExternalVisible := 'False'; ExternalWritable := 'False'} : Bool;   // HMICmd
      HMICmdResetCurrentLimit { ExternalAccessible := 'False'; ExternalVisible := 'False'; ExternalWritable := 'False'} : Bool;   // HMICmd
      HMICmdResetUndVolt { ExternalAccessible := 'False'; ExternalVisible := 'False'; ExternalWritable := 'False'} : Bool;   // HMICmd
      HMICmdResetShortCirc { ExternalAccessible := 'False'; ExternalVisible := 'False'; ExternalWritable := 'False'} : Bool;   // HMICmd
      HMICmdResetSystError { ExternalAccessible := 'False'; ExternalVisible := 'False'; ExternalWritable := 'False'} : Bool;   // HMICmd
      HMICmdTrsf { ExternalAccessible := 'False'; ExternalVisible := 'False'; ExternalWritable := 'False'} : Bool;   // HMICmd
      HMICmdSpareBit10 { ExternalAccessible := 'False'; ExternalVisible := 'False'; ExternalWritable := 'False'} : Bool;   // HMICmd
      HMICmdSpareBit11 { ExternalAccessible := 'False'; ExternalVisible := 'False'; ExternalWritable := 'False'} : Bool;   // HMICmd
      HMICmdSpareBit12 { ExternalAccessible := 'False'; ExternalVisible := 'False'; ExternalWritable := 'False'} : Bool;   // HMICmd
      HMICmdSpareBit13 { ExternalAccessible := 'False'; ExternalVisible := 'False'; ExternalWritable := 'False'} : Bool;   // HMICmd
      HMICmdSpareBit14 { ExternalAccessible := 'False'; ExternalVisible := 'False'; ExternalWritable := 'False'} : Bool;   // HMICmd
      HMICmdSpareBit15 { ExternalAccessible := 'False'; ExternalVisible := 'False'; ExternalWritable := 'False'} : Bool;   // HMICmd
      C_LocalResetOFF { ExternalAccessible := 'False'; ExternalVisible := 'False'; ExternalWritable := 'False'} : Bool;   // Config Local reset
      C_LocalResetBlown { ExternalAccessible := 'False'; ExternalVisible := 'False'; ExternalWritable := 'False'} : Bool;   // Config Local reset
      C_LocalResetExtOFF { ExternalAccessible := 'False'; ExternalVisible := 'False'; ExternalWritable := 'False'} : Bool;   // Config Local reset
      C_LocalResetCurrentLimit { ExternalAccessible := 'False'; ExternalVisible := 'False'; ExternalWritable := 'False'} : Bool;   // Config Local reset
      C_LocalResetUndVolt { ExternalAccessible := 'False'; ExternalVisible := 'False'; ExternalWritable := 'False'} : Bool;   // Config Local reset
      C_LocalResetShortCirc { ExternalAccessible := 'False'; ExternalVisible := 'False'; ExternalWritable := 'False'} : Bool;   // Config Local reset
      C_LocalResetSystError { ExternalAccessible := 'False'; ExternalVisible := 'False'; ExternalWritable := 'False'} : Bool;   // Config Local reset
      C_LocalResetSpareBit7 { ExternalAccessible := 'False'; ExternalVisible := 'False'; ExternalWritable := 'False'} : Bool;   // Config Local reset
      C_LocalResetSpareBit8 { ExternalAccessible := 'False'; ExternalVisible := 'False'; ExternalWritable := 'False'} : Bool;   // Config Local reset
      C_LocalResetSpareBit9 { ExternalAccessible := 'False'; ExternalVisible := 'False'; ExternalWritable := 'False'} : Bool;   // Config Local reset
      C_LocalResetSpareBit10 { ExternalAccessible := 'False'; ExternalVisible := 'False'; ExternalWritable := 'False'} : Bool;   // Config Local reset
      C_LocalResetSpareBit11 { ExternalAccessible := 'False'; ExternalVisible := 'False'; ExternalWritable := 'False'} : Bool;   // Config Local reset
      C_LocalResetSpareBit12 { ExternalAccessible := 'False'; ExternalVisible := 'False'; ExternalWritable := 'False'} : Bool;   // Config Local reset
      C_LocalResetSpareBit13 { ExternalAccessible := 'False'; ExternalVisible := 'False'; ExternalWritable := 'False'} : Bool;   // Config Local reset
      C_LocalResetSpareBit14 { ExternalAccessible := 'False'; ExternalVisible := 'False'; ExternalWritable := 'False'} : Bool;   // Config Local reset
      C_LocalResetSpareBit15 { ExternalAccessible := 'False'; ExternalVisible := 'False'; ExternalWritable := 'False'} : Bool;   // Config Local reset
      FuseState_Bit0 { ExternalAccessible := 'False'; ExternalVisible := 'False'; ExternalWritable := 'False'} : Bool;   // Fuse Status: status bit 0 (to be used together with bit 1)
      FuseState_Bit1 { ExternalAccessible := 'False'; ExternalVisible := 'False'; ExternalWritable := 'False'} : Bool;   // Fuse Status: status bit 1 (to be used together with bit 0)
      FuseState_BitReserve { ExternalAccessible := 'False'; ExternalVisible := 'False'; ExternalWritable := 'False'} : Bool;   // Fuse Status: Reserve
      FuseState_BitNewMod { ExternalAccessible := 'False'; ExternalVisible := 'False'; ExternalWritable := 'False'} : Bool;   // Fuse Status: New module on Bus
      FuseState_BitCurWarn { ExternalAccessible := 'False'; ExternalVisible := 'False'; ExternalWritable := 'False'} : Bool;   // Fuse Status: Current Warning (I > 0.9 * Inom)
      FuseState_BitUndVolt { ExternalAccessible := 'False'; ExternalVisible := 'False'; ExternalWritable := 'False'} : Bool;   // Fuse Status: Under voltage
      FuseState_BitShortCirc { ExternalAccessible := 'False'; ExternalVisible := 'False'; ExternalWritable := 'False'} : Bool;   // Fuse Status: Short circuit
      FuseState_BitSysError { ExternalAccessible := 'False'; ExternalVisible := 'False'; ExternalWritable := 'False'} : Bool;   // Fuse Status: System error
      CmdFuse { ExternalAccessible := 'False'; ExternalVisible := 'False'; ExternalWritable := 'False'} : Byte;   // output byte fuse
      GETInfo_InputVoltage { ExternalAccessible := 'False'; ExternalVisible := 'False'; ExternalWritable := 'False'} : Bool;   // GET Info Input Voltage
      GETInfo_OutputVoltage { ExternalAccessible := 'False'; ExternalVisible := 'False'; ExternalWritable := 'False'} : Bool;   // GET Info Output Voltage
      GETInfo_CurrentSetp { ExternalAccessible := 'False'; ExternalVisible := 'False'; ExternalWritable := 'False'} : Bool;   // GET Info Current setpoint
      GETInfo_ActCurrent { ExternalAccessible := 'False'; ExternalVisible := 'False'; ExternalWritable := 'False'} : Bool;   // GET Info Actual Current
      GETInfo_Curve { ExternalAccessible := 'False'; ExternalVisible := 'False'; ExternalWritable := 'False'} : Bool;   // GET Info Curve type
      Info_Busy { ExternalAccessible := 'False'; ExternalVisible := 'False'; ExternalWritable := 'False'} : Bool;   // Info Busy
      Info_InputVoltageOk { ExternalAccessible := 'False'; ExternalVisible := 'False'; ExternalWritable := 'False'} : Bool;   // Info Input Voltage OK
      Info_OutputVoltageOk { ExternalAccessible := 'False'; ExternalVisible := 'False'; ExternalWritable := 'False'} : Bool;   // Info Output Voltage OK
      Info_CurrentSetpOk { ExternalAccessible := 'False'; ExternalVisible := 'False'; ExternalWritable := 'False'} : Bool;   // Info Current setpoint OK
      Info_ActCurrentOk { ExternalAccessible := 'False'; ExternalVisible := 'False'; ExternalWritable := 'False'} : Bool;   // Info Actual Current OK
      Info_CurveOk { ExternalAccessible := 'False'; ExternalVisible := 'False'; ExternalWritable := 'False'} : Bool;   // Info Curve type OK
      ValueInfo_InputVoltage { ExternalAccessible := 'False'; ExternalVisible := 'False'; ExternalWritable := 'False'} : DWord;   // Calculate value Input Voltage
      ValueInfo_OutputVoltage { ExternalAccessible := 'False'; ExternalVisible := 'False'; ExternalWritable := 'False'} : DWord;   // Calculate value Output Voltage
      ValueInfo_CurrentSetp { ExternalAccessible := 'False'; ExternalVisible := 'False'; ExternalWritable := 'False'} : DWord;   // Calculate value Current setpoint
      ValueInfo_ActCurrent { ExternalAccessible := 'False'; ExternalVisible := 'False'; ExternalWritable := 'False'} : DWord;   // Calculate value Actual Current
      ValueInfo_Curve { ExternalAccessible := 'False'; ExternalVisible := 'False'; ExternalWritable := 'False'} : DWord;   // CHAR Curve type
      ResetInfoBusy { ExternalAccessible := 'False'; ExternalVisible := 'False'; ExternalWritable := 'False'} : Bool;   // Reset signal Info busy
      DBnr { ExternalAccessible := 'False'; ExternalVisible := 'False'; ExternalWritable := 'False'} : Int;   // HMI DB number
      RDREC_REQ { ExternalAccessible := 'False'; ExternalVisible := 'False'; ExternalWritable := 'False'} : Bool;   // Read function
      RDREC_INDEX { ExternalAccessible := 'False'; ExternalVisible := 'False'; ExternalWritable := 'False'} : DWord;   // Read function
      RDREC_MLEN { ExternalAccessible := 'False'; ExternalVisible := 'False'; ExternalWritable := 'False'} : Word;   // Read function
      RDREC_Record { ExternalAccessible := 'False'; ExternalVisible := 'False'; ExternalWritable := 'False'} : DWord;   // Read function
      RDREC_Valid { ExternalAccessible := 'False'; ExternalVisible := 'False'; ExternalWritable := 'False'} : Bool;   // Read function
      RDREC_Busy { ExternalAccessible := 'False'; ExternalVisible := 'False'; ExternalWritable := 'False'} : Bool;   // Read function
      RDREC_Error { ExternalAccessible := 'False'; ExternalVisible := 'False'; ExternalWritable := 'False'} : Bool;   // Read function
      RDREC_Status { ExternalAccessible := 'False'; ExternalVisible := 'False'; ExternalWritable := 'False'} : DWord;   // Read function
      RDREC_LEN { ExternalAccessible := 'False'; ExternalVisible := 'False'; ExternalWritable := 'False'} : Word;   // Read function
      InfoNotUptoDate { ExternalAccessible := 'False'; ExternalVisible := 'False'; ExternalWritable := 'False'} : Bool;   // The info (data from the fuse) is not more up-to-date
      Edge001 { ExternalAccessible := 'False'; ExternalVisible := 'False'; ExternalWritable := 'False'} : Bool;   // Edge
   END_VAR
   VAR
      RDREC { ExternalAccessible := 'False'; ExternalVisible := 'False'; ExternalWritable := 'False'} : RDREC;   // Read info from LoccBox Fuse
   END_VAR
   VAR DB_SPECIFIC
      TimerInit { ExternalAccessible := 'False'; ExternalVisible := 'False'; ExternalWritable := 'False'} : TON_TIME;   // Timer
      TimerBusy { ExternalAccessible := 'False'; ExternalVisible := 'False'; ExternalWritable := 'False'} : TON_TIME;   // Timer
      TimerRestart { ExternalAccessible := 'False'; ExternalVisible := 'False'; ExternalWritable := 'False'} : TON_TIME;   // Timer
   END_VAR
   VAR_TEMP
      TempINT : Int;
      TempDINT : DInt;
      TempDWORD : DWord;
      TempREAL : Real;
   END_VAR
   VAR_TEMP   // added for the SCL form of the ladder/FBD networks
      _w1 : Bool;
   END_VAR
BEGIN

NETWORK
TITLE = **** 1 - Inputs **** DB number
// DB number
      L     DINO;
      T     #DBnr;

NETWORK
TITLE = **** 1 - Inputs **** Alarm class
// Alarm class
// Alarm class = D
      L     #I_AlarmClass;
      L     'D';
      ==I;
      =     #AlarmClass_D;

// Alarm class = C
      L     #I_AlarmClass;
      L     'C';
      ==I;
      =     #AlarmClass_C;

// Alarm class = B
      L     #I_AlarmClass;
      L     'B';
      ==I;
      =     #AlarmClass_B;

// Alarm class = A
      AN    #AlarmClass_B;
      AN    #AlarmClass_C;
      AN    #AlarmClass_D;
      =     #AlarmClass_A;


REGION Network 3: **** 1 - Inputs **** Fuse Status: status bit 0 (to be used together with bit 1)
   // Bit Fuse Status: status bit 0 (to be used together with bit 1)
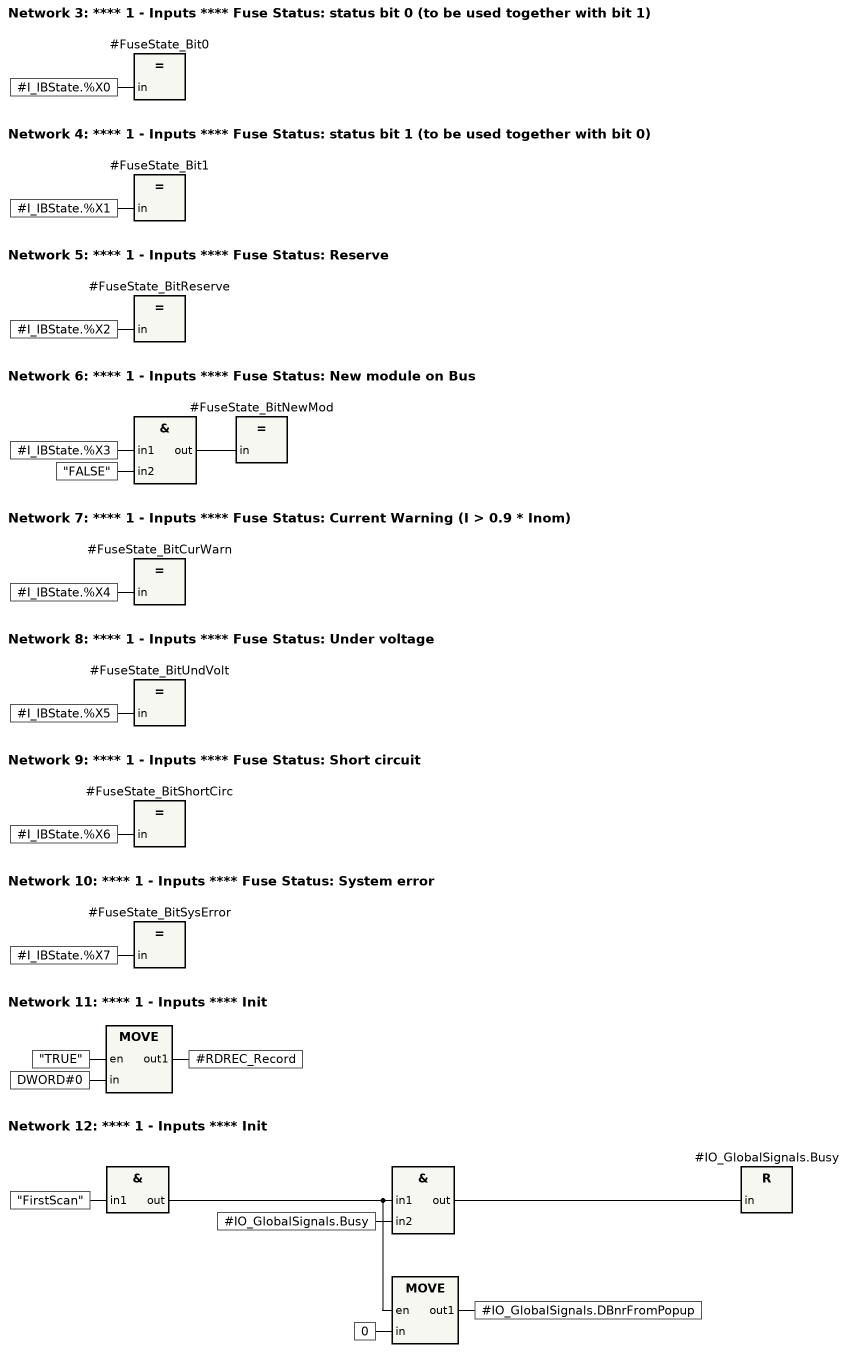
   #FuseState_Bit0 := #I_IBState.%X0;
END_REGION

REGION Network 4: **** 1 - Inputs **** Fuse Status: status bit 1 (to be used together with bit 0)
   // Fuse Status: status bit 1 (to be used together with bit 0)
   #FuseState_Bit1 := #I_IBState.%X1;
END_REGION

REGION Network 5: **** 1 - Inputs **** Fuse Status: Reserve
   // Fuse Status: Reserve
   #FuseState_BitReserve := #I_IBState.%X2;
END_REGION

REGION Network 6: **** 1 - Inputs **** Fuse Status: New module on Bus
   // Fuse Status: New module on Bus
   #FuseState_BitNewMod := #I_IBState.%X3 AND "FALSE";
END_REGION

REGION Network 7: **** 1 - Inputs **** Fuse Status: Current Warning (I > 0.9 * Inom)
   // Fuse Status: Current Warning (I > 0.9 * Inom)
   #FuseState_BitCurWarn := #I_IBState.%X4;
END_REGION

REGION Network 8: **** 1 - Inputs **** Fuse Status: Under voltage
   // Fuse Status: Under voltage
   #FuseState_BitUndVolt := #I_IBState.%X5;
END_REGION

REGION Network 9: **** 1 - Inputs **** Fuse Status: Short circuit
   // Fuse Status: Short circuit
   #FuseState_BitShortCirc := #I_IBState.%X6;
END_REGION

REGION Network 10: **** 1 - Inputs **** Fuse Status: System error
   // Fuse Status: System error
   #FuseState_BitSysError := #I_IBState.%X7;
END_REGION

REGION Network 11: **** 1 - Inputs **** Init
   // Init
   IF "TRUE" THEN #RDREC_Record := DWORD#0; END_IF;
END_REGION

REGION Network 12: **** 1 - Inputs **** Init
   // Init
   IF "FirstScan" AND #IO_GlobalSignals.Busy THEN #IO_GlobalSignals.Busy := FALSE; END_IF;
   IF "FirstScan" THEN #IO_GlobalSignals.DBnrFromPopup := 0; END_IF;
END_REGION

REGION Network 13: **** 1 - Inputs **** Init
   // Init
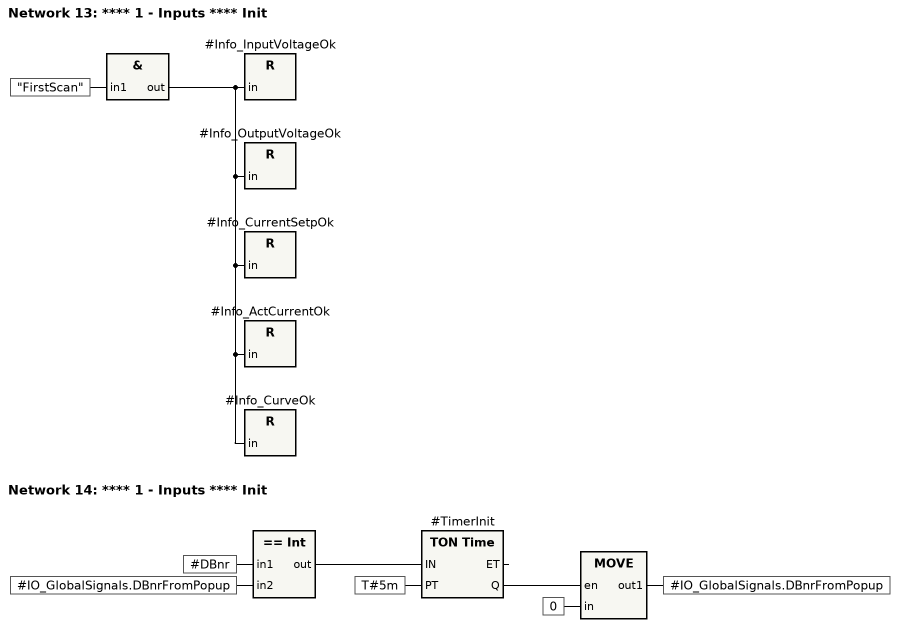
   IF "FirstScan" THEN
       #Info_InputVoltageOk := FALSE;
       #Info_OutputVoltageOk := FALSE;
       #Info_CurrentSetpOk := FALSE;
       #Info_ActCurrentOk := FALSE;
       #Info_CurveOk := FALSE;
   END_IF;
END_REGION

REGION Network 14: **** 1 - Inputs **** Init
   // Init
   #TimerInit(IN := #DBnr = #IO_GlobalSignals.DBnrFromPopup, PT := T#5m);   // TON
   IF #TimerInit.Q THEN #IO_GlobalSignals.DBnrFromPopup := 0; END_IF;
END_REGION

REGION Network 15: **** 1 - Inputs **** Used to define if for this installation a status is alarm or warning
   // Extract the configuration
   // Used to define if for this installation a status is alarm or warning
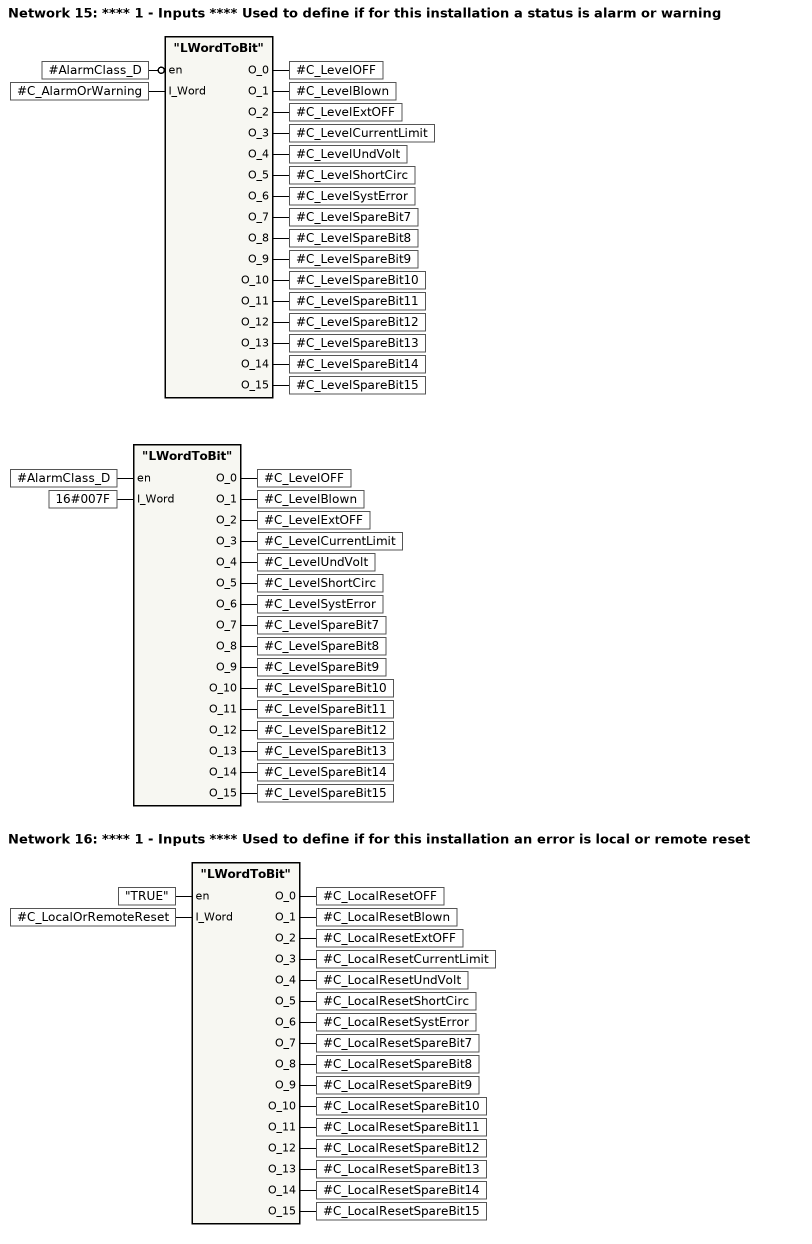
   IF NOT #AlarmClass_D THEN
       "LWordToBit"(I_Word := #C_AlarmOrWarning,
                    O_0 => #C_LevelOFF,
                    O_1 => #C_LevelBlown,
                    O_2 => #C_LevelExtOFF,
                    O_3 => #C_LevelCurrentLimit,
                    O_4 => #C_LevelUndVolt,
                    O_5 => #C_LevelShortCirc,
                    O_6 => #C_LevelSystError,
                    O_7 => #C_LevelSpareBit7,
                    O_8 => #C_LevelSpareBit8,
                    O_9 => #C_LevelSpareBit9,
                    O_10 => #C_LevelSpareBit10,
                    O_11 => #C_LevelSpareBit11,
                    O_12 => #C_LevelSpareBit12,
                    O_13 => #C_LevelSpareBit13,
                    O_14 => #C_LevelSpareBit14,
                    O_15 => #C_LevelSpareBit15);
   END_IF;
   IF #AlarmClass_D THEN
       "LWordToBit"(I_Word := 16#007F,
                    O_0 => #C_LevelOFF,
                    O_1 => #C_LevelBlown,
                    O_2 => #C_LevelExtOFF,
                    O_3 => #C_LevelCurrentLimit,
                    O_4 => #C_LevelUndVolt,
                    O_5 => #C_LevelShortCirc,
                    O_6 => #C_LevelSystError,
                    O_7 => #C_LevelSpareBit7,
                    O_8 => #C_LevelSpareBit8,
                    O_9 => #C_LevelSpareBit9,
                    O_10 => #C_LevelSpareBit10,
                    O_11 => #C_LevelSpareBit11,
                    O_12 => #C_LevelSpareBit12,
                    O_13 => #C_LevelSpareBit13,
                    O_14 => #C_LevelSpareBit14,
                    O_15 => #C_LevelSpareBit15);
   END_IF;
END_REGION

REGION Network 16: **** 1 - Inputs **** Used to define if for this installation an error is local or remote reset
   // Extract the configuration
   // Used to define if for this installation an error is local or remote reset
   IF "TRUE" THEN
       "LWordToBit"(I_Word := #C_LocalOrRemoteReset,
                    O_0 => #C_LocalResetOFF,
                    O_1 => #C_LocalResetBlown,
                    O_2 => #C_LocalResetExtOFF,
                    O_3 => #C_LocalResetCurrentLimit,
                    O_4 => #C_LocalResetUndVolt,
                    O_5 => #C_LocalResetShortCirc,
                    O_6 => #C_LocalResetSystError,
                    O_7 => #C_LocalResetSpareBit7,
                    O_8 => #C_LocalResetSpareBit8,
                    O_9 => #C_LocalResetSpareBit9,
                    O_10 => #C_LocalResetSpareBit10,
                    O_11 => #C_LocalResetSpareBit11,
                    O_12 => #C_LocalResetSpareBit12,
                    O_13 => #C_LocalResetSpareBit13,
                    O_14 => #C_LocalResetSpareBit14,
                    O_15 => #C_LocalResetSpareBit15);
   END_IF;
END_REGION

REGION Network 17: **** 1 - Inputs **** HMI Command
   // Extract the HMI command bit
   // Command bit from HMI
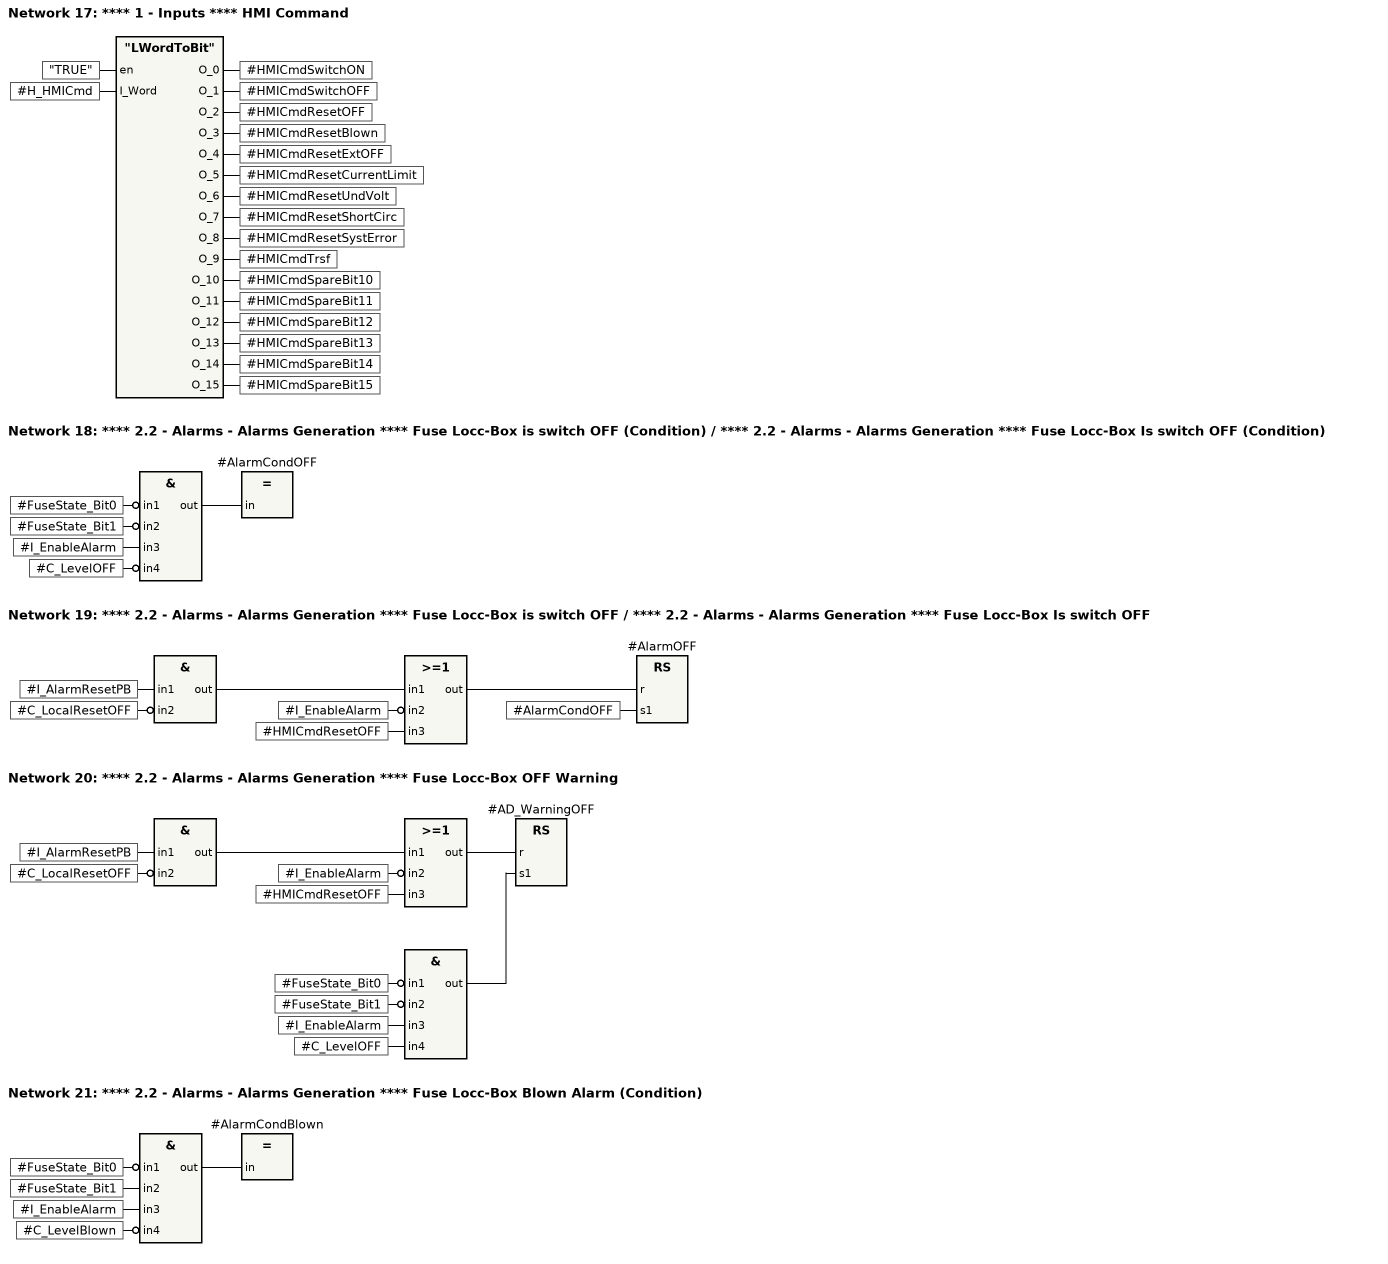
   IF "TRUE" THEN
       "LWordToBit"(I_Word := #H_HMICmd,
                    O_0 => #HMICmdSwitchON,
                    O_1 => #HMICmdSwitchOFF,
                    O_2 => #HMICmdResetOFF,
                    O_3 => #HMICmdResetBlown,
                    O_4 => #HMICmdResetExtOFF,
                    O_5 => #HMICmdResetCurrentLimit,
                    O_6 => #HMICmdResetUndVolt,
                    O_7 => #HMICmdResetShortCirc,
                    O_8 => #HMICmdResetSystError,
                    O_9 => #HMICmdTrsf,
                    O_10 => #HMICmdSpareBit10,
                    O_11 => #HMICmdSpareBit11,
                    O_12 => #HMICmdSpareBit12,
                    O_13 => #HMICmdSpareBit13,
                    O_14 => #HMICmdSpareBit14,
                    O_15 => #HMICmdSpareBit15);
   END_IF;
END_REGION

REGION Network 18: **** 2.2 - Alarms - Alarms Generation **** Fuse Locc-Box is switch OFF (Condition) / **** 2.2 - Alarms - Alarms Generation **** Fuse Locc-Box Is switch OFF (Condition)
   // Condition for the Alarm
   #AlarmCondOFF := NOT #FuseState_Bit0 AND NOT #FuseState_Bit1 AND #I_EnableAlarm AND NOT #C_LevelOFF;
END_REGION

REGION Network 19: **** 2.2 - Alarms - Alarms Generation **** Fuse Locc-Box is switch OFF / **** 2.2 - Alarms - Alarms Generation **** Fuse Locc-Box Is switch OFF
   // Memorisation of the Alarm
   IF (#I_AlarmResetPB AND NOT #C_LocalResetOFF) OR NOT #I_EnableAlarm OR #HMICmdResetOFF THEN
       #AlarmOFF := FALSE;   // RS flip-flop
   END_IF;
   IF #AlarmCondOFF THEN #AlarmOFF := TRUE; END_IF;
END_REGION

REGION Network 20: **** 2.2 - Alarms - Alarms Generation **** Fuse Locc-Box OFF Warning
   // Memorisation of the Alarm
   IF (#I_AlarmResetPB AND NOT #C_LocalResetOFF) OR NOT #I_EnableAlarm OR #HMICmdResetOFF THEN
       #AD_WarningOFF := FALSE;   // RS flip-flop
   END_IF;
   IF NOT #FuseState_Bit0 AND NOT #FuseState_Bit1 AND #I_EnableAlarm AND #C_LevelOFF THEN
       #AD_WarningOFF := TRUE;
   END_IF;
END_REGION

REGION Network 21: **** 2.2 - Alarms - Alarms Generation **** Fuse Locc-Box Blown Alarm (Condition)
   // Condition for the Alarm
   #AlarmCondBlown := NOT #FuseState_Bit0 AND #FuseState_Bit1 AND #I_EnableAlarm AND NOT #C_LevelBlown;
END_REGION

REGION Network 22: **** 2.2 - Alarms - Alarms Generation **** Fuse Locc-Box Blown Alarm
   // Memorisation of the Alarm
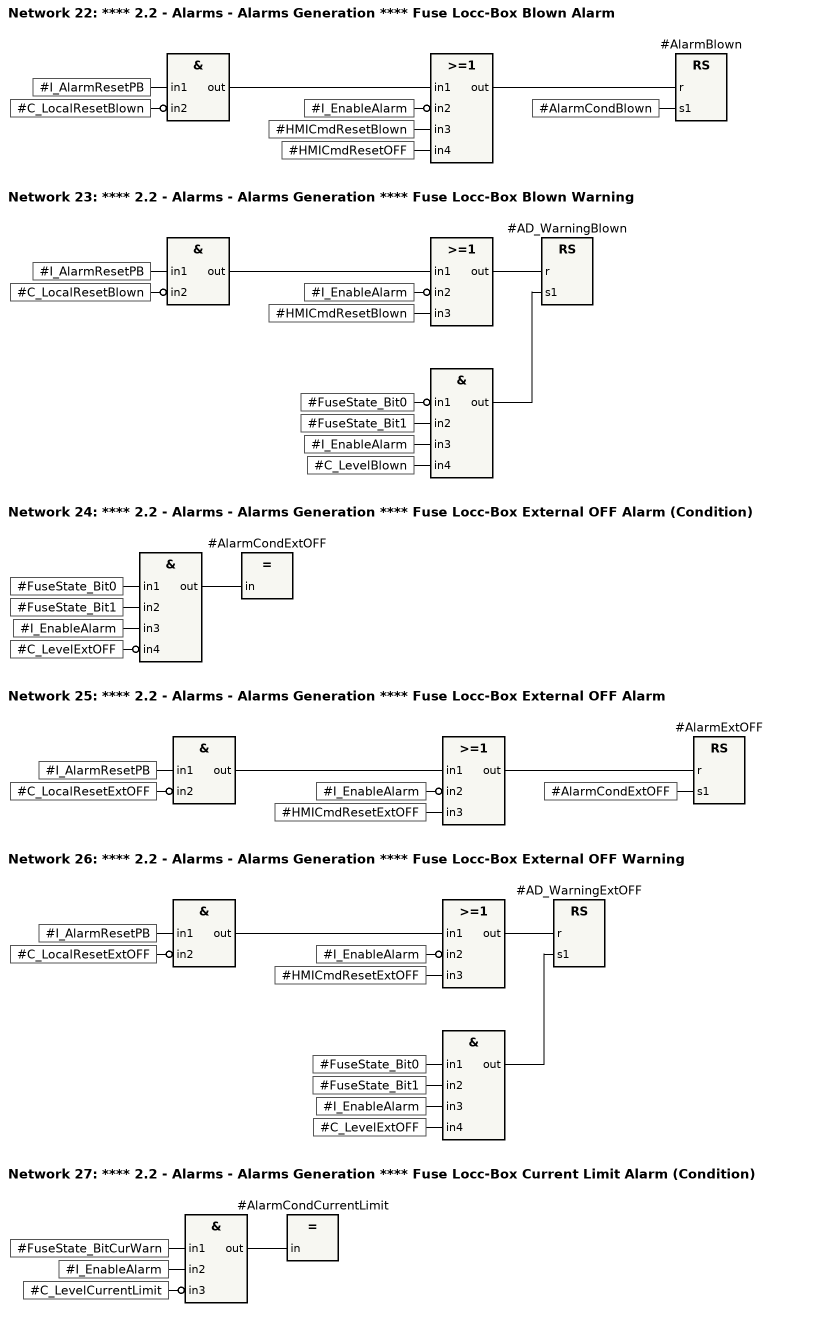
   IF (#I_AlarmResetPB AND NOT #C_LocalResetBlown) OR NOT #I_EnableAlarm OR #HMICmdResetBlown OR #HMICmdResetOFF THEN
       #AlarmBlown := FALSE;   // RS flip-flop
   END_IF;
   IF #AlarmCondBlown THEN #AlarmBlown := TRUE; END_IF;
END_REGION

REGION Network 23: **** 2.2 - Alarms - Alarms Generation **** Fuse Locc-Box Blown Warning
   // Memorisation of the Alarm
   IF (#I_AlarmResetPB AND NOT #C_LocalResetBlown) OR NOT #I_EnableAlarm OR #HMICmdResetBlown THEN
       #AD_WarningBlown := FALSE;   // RS flip-flop
   END_IF;
   IF NOT #FuseState_Bit0 AND #FuseState_Bit1 AND #I_EnableAlarm AND #C_LevelBlown THEN
       #AD_WarningBlown := TRUE;
   END_IF;
END_REGION

REGION Network 24: **** 2.2 - Alarms - Alarms Generation **** Fuse Locc-Box External OFF Alarm (Condition)
   // Condition for the Alarm
   #AlarmCondExtOFF := #FuseState_Bit0 AND #FuseState_Bit1 AND #I_EnableAlarm AND NOT #C_LevelExtOFF;
END_REGION

REGION Network 25: **** 2.2 - Alarms - Alarms Generation **** Fuse Locc-Box External OFF Alarm
   // Memorisation of the Alarm
   IF (#I_AlarmResetPB AND NOT #C_LocalResetExtOFF) OR NOT #I_EnableAlarm OR #HMICmdResetExtOFF THEN
       #AlarmExtOFF := FALSE;   // RS flip-flop
   END_IF;
   IF #AlarmCondExtOFF THEN #AlarmExtOFF := TRUE; END_IF;
END_REGION

REGION Network 26: **** 2.2 - Alarms - Alarms Generation **** Fuse Locc-Box External OFF Warning
   // Memorisation of the Alarm
   IF (#I_AlarmResetPB AND NOT #C_LocalResetExtOFF) OR NOT #I_EnableAlarm OR #HMICmdResetExtOFF THEN
       #AD_WarningExtOFF := FALSE;   // RS flip-flop
   END_IF;
   IF #FuseState_Bit0 AND #FuseState_Bit1 AND #I_EnableAlarm AND #C_LevelExtOFF THEN
       #AD_WarningExtOFF := TRUE;
   END_IF;
END_REGION

REGION Network 27: **** 2.2 - Alarms - Alarms Generation **** Fuse Locc-Box Current Limit Alarm (Condition)
   // Condition for the Alarm
   #AlarmCondCurrentLimit := #FuseState_BitCurWarn AND #I_EnableAlarm AND NOT #C_LevelCurrentLimit;
END_REGION

REGION Network 28: **** 2.2 - Alarms - Alarms Generation **** Fuse Locc-Box Current Limit Alarm
   // Memorisation of the Alarm
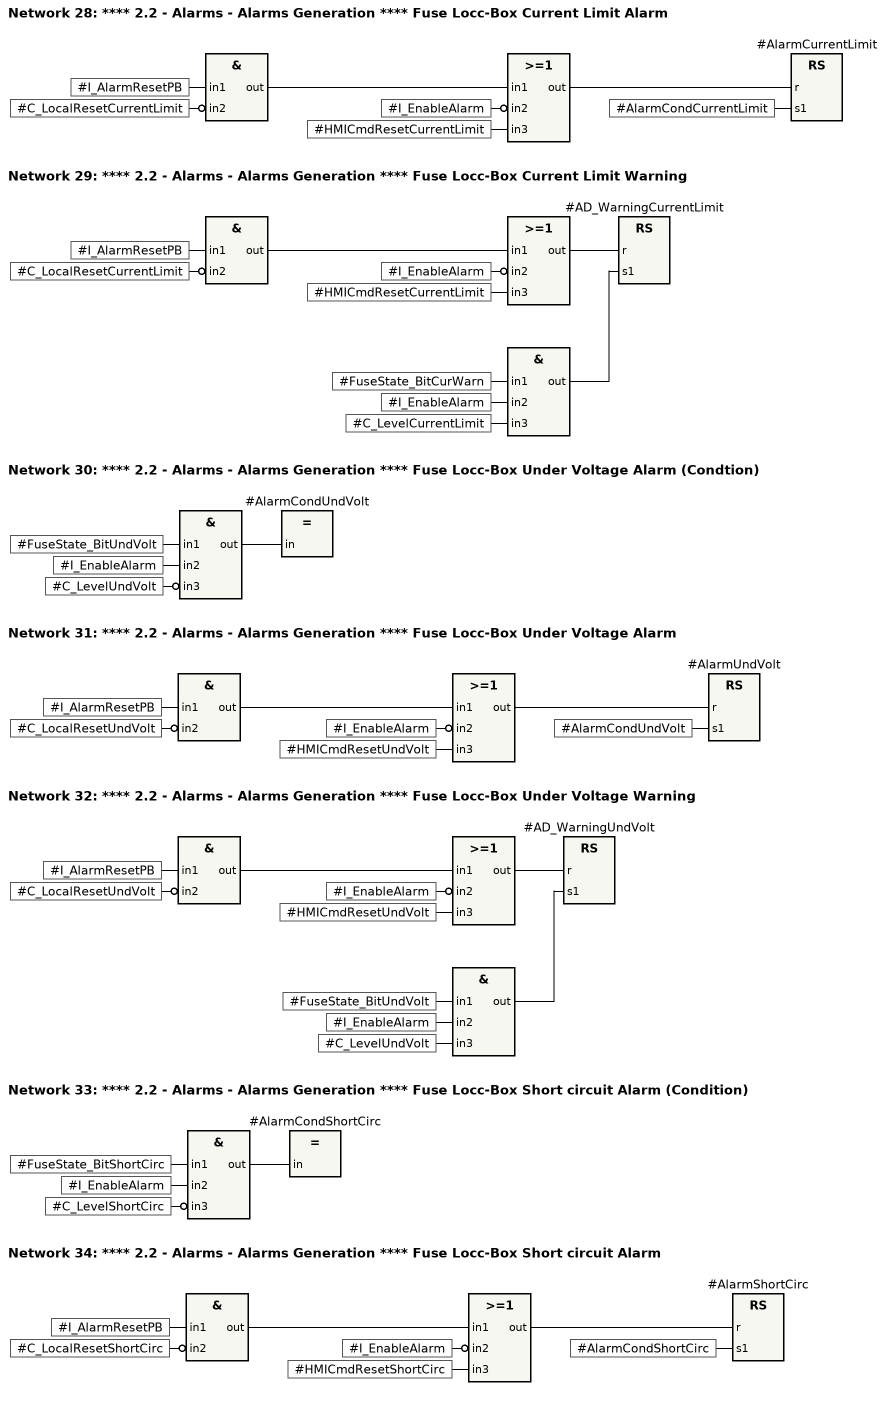
   IF (#I_AlarmResetPB AND NOT #C_LocalResetCurrentLimit) OR NOT #I_EnableAlarm OR #HMICmdResetCurrentLimit THEN
       #AlarmCurrentLimit := FALSE;   // RS flip-flop
   END_IF;
   IF #AlarmCondCurrentLimit THEN #AlarmCurrentLimit := TRUE; END_IF;
END_REGION

REGION Network 29: **** 2.2 - Alarms - Alarms Generation **** Fuse Locc-Box Current Limit Warning
   // Memorisation of the Alarm
   IF (#I_AlarmResetPB AND NOT #C_LocalResetCurrentLimit) OR NOT #I_EnableAlarm OR #HMICmdResetCurrentLimit THEN
       #AD_WarningCurrentLimit := FALSE;   // RS flip-flop
   END_IF;
   IF #FuseState_BitCurWarn AND #I_EnableAlarm AND #C_LevelCurrentLimit THEN
       #AD_WarningCurrentLimit := TRUE;
   END_IF;
END_REGION

REGION Network 30: **** 2.2 - Alarms - Alarms Generation **** Fuse Locc-Box Under Voltage Alarm (Condtion)
   // Condition for the Alarm
   #AlarmCondUndVolt := #FuseState_BitUndVolt AND #I_EnableAlarm AND NOT #C_LevelUndVolt;
END_REGION

REGION Network 31: **** 2.2 - Alarms - Alarms Generation **** Fuse Locc-Box Under Voltage Alarm
   // Memorisation of the Alarm
   IF (#I_AlarmResetPB AND NOT #C_LocalResetUndVolt) OR NOT #I_EnableAlarm OR #HMICmdResetUndVolt THEN
       #AlarmUndVolt := FALSE;   // RS flip-flop
   END_IF;
   IF #AlarmCondUndVolt THEN #AlarmUndVolt := TRUE; END_IF;
END_REGION

REGION Network 32: **** 2.2 - Alarms - Alarms Generation **** Fuse Locc-Box Under Voltage Warning
   // Memorisation of the Alarm
   IF (#I_AlarmResetPB AND NOT #C_LocalResetUndVolt) OR NOT #I_EnableAlarm OR #HMICmdResetUndVolt THEN
       #AD_WarningUndVolt := FALSE;   // RS flip-flop
   END_IF;
   IF #FuseState_BitUndVolt AND #I_EnableAlarm AND #C_LevelUndVolt THEN #AD_WarningUndVolt := TRUE; END_IF;
END_REGION

